LIN {X 0.066,Y -342.282,Z 1020.656,A 0.000,B 0.000,C 90.000,E1 118.103} C_DIS
LIN {X 0.176,Y -355.213,Z 1020.641,A 0.000,B 0.000,C 90.000,E1 115.335} C_DIS
LIN {X 0.119,Y -368.001,Z 1020.628,A 0.000,B 0.000,C 90.000,E1 112.950} C_DIS
LIN {X 0.098,Y -382.100,Z 1020.615,A 0.000,B 0.000,C 90.000,E1 110.610} C_DIS
LIN {X -0.206,Y -397.609,Z 1020.602,A 0.000,B 0.000,C 90.000,E1 108.362} C_DIS
LIN {X 0.126,Y -414.640,Z 1020.589,A 0.000,B 0.000,C 90.000,E1 106.079} C_DIS
LIN {X -0.157,Y -433.313,Z 1020.577,A 0.000,B 0.000,C 90.000,E1 103.939} C_DIS
LIN {X 0.189,Y -453.249,Z 1020.566,A 0.000,B 0.000,C 90.000,E1 101.827} C_DIS
LIN {X -0.120,Y -466.020,Z 1020.559,A 0.000,B 0.000,C 90.000,E1 100.658} C_DIS
LIN {X -0.093,Y -468.376,Z 1020.558,A 0.000,B 0.000,C 90.000,E1 100.423} C_DIS
LIN {X -0.148,Y -470.162,Z 1020.557,A 0.000,B 0.000,C 90.000,E1 100.197} C_DIS
LIN {X 0.167,Y -471.645,Z 1020.555,A 0.000,B 0.000,C 90.000,E1 99.905} C_DIS
LIN {X 0.018,Y -472.751,Z 1020.554,A 0.000,B 0.000,C 90.000,E1 99.670} C_DIS
LIN {X 0.125,Y -474.065,Z 1020.551,A 0.000,B 0.000,C 90.000,E1 99.151} C_DIS
LIN {X -0.156,Y -474.365,Z 1020.548,A 0.000,B 0.000,C 90.000,E1 98.681} C_DIS
LIN {X -0.034,Y -473.699,Z 1020.545,A 0.000,B 0.000,C 90.000,E1 98.163} C_DIS
LIN {X 0.093,Y -471.967,Z 1020.543,A 0.000,B 0.000,C 90.000,E1 97.644} C_DIS
LIN {X -0.049,Y -470.604,Z 1020.541,A 0.000,B 0.000,C 90.000,E1 97.409} C_DIS
LIN {X 0.009,Y -458.360,Z 1020.531,A 0.000,B 0.000,C 90.000,E1 95.625} C_DIS
LIN {X -0.178,Y -445.807,Z 1020.521,A 0.000,B 0.000,C 90.000,E1 93.841} C_DIS
LIN {X -0.035,Y -427.414,Z 1020.505,A 0.000,B 0.000,C 90.000,E1 90.917} C_DIS
LIN {X -0.048,Y -411.025,Z 1020.489,A 0.000,B 0.000,C 90.000,E1 87.936} C_DIS
LIN {X -0.010,Y -402.181,Z 1020.479,A 0.000,B 0.000,C 90.000,E1 86.274} C_DIS
LIN {X -0.112,Y -393.138,Z 1020.470,A 0.000,B 0.000,C 90.000,E1 84.609} C_DIS
LIN {X 0.091,Y -383.865,Z 1020.461,A 0.000,B 0.000,C 90.000,E1 82.875} C_DIS
LIN {X 0.119,Y -376.009,Z 1020.453,A 0.000,B 0.000,C 90.000,E1 81.432} C_DIS
LIN {X 0.047,Y -364.517,Z 1020.441,A 0.000,B 0.000,C 90.000,E1 79.398} C_DIS
LIN {X -0.187,Y -352.885,Z 1020.430,A 0.000,B 0.000,C 90.000,E1 77.353} C_DIS
LIN {X 0.067,Y -338.162,Z 1020.414,A 0.000,B 0.000,C 90.000,E1 74.574} C_DIS
LIN {X -0.175,Y -325.593,Z 1020.401,A 0.000,B 0.000,C 90.000,E1 72.127} C_DIS
LIN {X -0.035,Y -314.862,Z 1020.388,A 0.000,B 0.000,C 90.000,E1 69.880} C_DIS
LIN {X -0.110,Y -301.369,Z 1020.372,A 0.000,B 0.000,C 90.000,E1 66.975} C_DIS
LIN {X -0.154,Y -291.133,Z 1020.359,A 0.000,B 0.000,C 90.000,E1 64.665} C_DIS
LIN {X -0.052,Y -281.166,Z 1020.346,A 0.000,B 0.000,C 90.000,E1 62.281} C_DIS
LIN {X -0.099,Y -269.958,Z 1020.331,A 0.000,B 0.000,C 90.000,E1 59.537} C_DIS
LIN {X 0.078,Y -260.291,Z 1020.317,A 0.000,B 0.000,C 90.000,E1 57.041} C_DIS
LIN {X -0.018,Y -249.657,Z 1020.301,A 0.000,B 0.000,C 90.000,E1 54.196} C_DIS
LIN {X 0.045,Y -238.282,Z 1020.283,A 0.000,B 0.000,C 90.000,E1 50.884} C_DIS
LIN {X -0.116,Y -227.694,Z 1020.264,A 0.000,B 0.000,C 90.000,E1 47.553} C_DIS
LIN {X 0.123,Y -218.751,Z 1020.247,A 0.000,B 0.000,C 90.000,E1 44.433} C_DIS
LIN {X 0.004,Y -210.152,Z 1020.230,A 0.000,B 0.000,C 90.000,E1 41.353} C_DIS
LIN {X 0.040,Y -202.163,Z 1020.212,A 0.000,B 0.000,C 90.000,E1 38.177} C_DIS
LIN {X -0.039,Y -194.792,Z 1020.194,A 0.000,B 0.000,C 90.000,E1 34.978} C_DIS
LIN {X 0.070,Y -188.093,Z 1020.176,A 0.000,B 0.000,C 90.000,E1 31.671} C_DIS
LIN {X 0.036,Y -182.287,Z 1020.158,A 0.000,B 0.000,C 90.000,E1 28.359} C_DIS
LIN {X -0.071,Y -177.205,Z 1020.139,A 0.000,B 0.000,C 90.000,E1 25.027} C_DIS
LIN {X 0.031,Y -172.984,Z 1020.120,A 0.000,B 0.000,C 90.000,E1 21.589} C_DIS
LIN {X -0.060,Y -169.399,Z 1020.101,A 0.000,B 0.000,C 90.000,E1 18.181} C_DIS
LIN {X -0.011,Y -165.911,Z 1020.077,A 0.000,B 0.000,C 90.000,E1 13.828} C_DIS
LIN {X 0.025,Y -163.211,Z 1020.048,A 0.000,B 0.000,C 90.000,E1 8.568} C_DIS
LIN {X 0.015,Y -164.093,Z 1019.953,A 0.000,B 0.000,C 90.000,E1 351.602} C_DIS
LIN {X 0.009,Y -167.296,Z 1019.924,A 0.000,B 0.000,C 90.000,E1 346.353} C_DIS
LIN {X 0.037,Y -171.068,Z 1019.900,A 0.000,B 0.000,C 90.000,E1 342.000} C_DIS
LIN {X -0.079,Y -174.981,Z 1019.881,A 0.000,B 0.000,C 90.000,E1 338.592} C_DIS
LIN {X -0.001,Y -179.715,Z 1019.862,A 0.000,B 0.000,C 90.000,E1 335.153} C_DIS
LIN {X 0.024,Y -185.257,Z 1019.843,A 0.000,B 0.000,C 90.000,E1 331.769} C_DIS
LIN {X -0.041,Y -191.575,Z 1019.825,A 0.000,B 0.000,C 90.000,E1 328.456} C_DIS
LIN {X -0.078,Y -198.576,Z 1019.806,A 0.000,B 0.000,C 90.000,E1 325.182} C_DIS
LIN {X -0.040,Y -207.196,Z 1019.786,A 0.000,B 0.000,C 90.000,E1 321.537} C_DIS
LIN {X 0.037,Y -216.493,Z 1019.766,A 0.000,B 0.000,C 90.000,E1 317.957} C_DIS
LIN {X 0.107,Y -225.454,Z 1019.749,A 0.000,B 0.000,C 90.000,E1 314.838} C_DIS
LIN {X -0.021,Y -234.071,Z 1019.734,A 0.000,B 0.000,C 90.000,E1 312.204} C_DIS
LIN {X 0.094,Y -242.569,Z 1019.722,A 0.000,B 0.000,C 90.000,E1 309.930} C_DIS
LIN {X 0.056,Y -248.911,Z 1019.714,A 0.000,B 0.000,C 90.000,E1 308.463} C_DIS
LIN {X -0.034,Y -257.706,Z 1019.704,A 0.000,B 0.000,C 90.000,E1 306.664} C_DIS
LIN {X -0.168,Y -271.393,Z 1019.690,A 0.000,B 0.000,C 90.000,E1 304.199} C_DIS
LIN {X 0.040,Y -288.410,Z 1019.674,A 0.000,B 0.000,C 90.000,E1 301.386} C_DIS
LIN {X 0.130,Y -309.092,Z 1019.658,A 0.000,B 0.000,C 90.000,E1 298.359} C_DIS
LIN {X 0.007,Y -324.070,Z 1019.647,A 0.000,B 0.000,C 90.000,E1 296.437} C_DIS
LIN {X -0.043,Y -337.092,Z 1019.639,A 0.000,B 0.000,C 90.000,E1 294.951} C_DIS
LIN {X -0.147,Y -364.351,Z 1019.623,A 0.000,B 0.000,C 90.000,E1 292.206} C_DIS
LIN {X -0.138,Y -383.717,Z 1019.613,A 0.000,B 0.000,C 90.000,E1 290.429} C_DIS
LIN {X 0.093,Y -402.310,Z 1019.604,A 0.000,B 0.000,C 90.000,E1 288.725} C_DIS
LIN {X 0.012,Y -412.772,Z 1019.599,A 0.000,B 0.000,C 90.000,E1 287.764} C_DIS
LIN {X -0.146,Y -420.410,Z 1019.595,A 0.000,B 0.000,C 90.000,E1 287.040} C_DIS
LIN {X -0.161,Y -427.896,Z 1019.590,A 0.000,B 0.000,C 90.000,E1 286.260} C_DIS
LIN {X -0.164,Y -437.601,Z 1019.584,A 0.000,B 0.000,C 90.000,E1 285.190} C_DIS
LIN {X -0.089,Y -446.673,Z 1019.578,A 0.000,B 0.000,C 90.000,E1 284.120} C_DIS
LIN {X -0.014,Y -455.104,Z 1019.573,A 0.000,B 0.000,C 90.000,E1 283.063} C_DIS
LIN {X -0.114,Y -460.826,Z 1019.568,A 0.000,B 0.000,C 90.000,E1 282.299} C_DIS
LIN {X -0.161,Y -466.044,Z 1019.564,A 0.000,B 0.000,C 90.000,E1 281.535} C_DIS
LIN {X -0.261,Y -470.809,Z 1019.560,A 0.000,B 0.000,C 90.000,E1 280.782} C_DIS
LIN {X 0.241,Y -474.949,Z 1019.555,A 0.000,B 0.000,C 90.000,E1 279.962} C_DIS
LIN {X 0.228,Y -478.512,Z 1019.551,A 0.000,B 0.000,C 90.000,E1 279.208} C_DIS
LIN {X -0.101,Y -480.580,Z 1019.549,A 0.000,B 0.000,C 90.000,E1 278.746} C_DIS
LIN {X 0.128,Y -482.342,Z 1019.546,A 0.000,B 0.000,C 90.000,E1 278.219} C_DIS
LIN {X -0.010,Y -485.160,Z 1019.540,A 0.000,B 0.000,C 90.000,E1 277.239} C_DIS
LIN {X 0.176,Y -486.261,Z 1019.537,A 0.000,B 0.000,C 90.000,E1 276.720} C_DIS
LIN {X -0.113,Y -487.145,Z 1019.535,A 0.000,B 0.000,C 90.000,E1 276.258} C_DIS
LIN {X 0.088,Y -487.739,Z 1019.532,A 0.000,B 0.000,C 90.000,E1 275.739} C_DIS
LIN {X -0.193,Y -487.996,Z 1019.529,A 0.000,B 0.000,C 90.000,E1 275.277} C_DIS
LIN {X 0.015,Y -487.823,Z 1019.526,A 0.000,B 0.000,C 90.000,E1 274.759} C_DIS
LIN {X 0.184,Y -487.214,Z 1019.524,A 0.000,B 0.000,C 90.000,E1 274.245} C_DIS
LIN {X -0.096,Y -486.033,Z 1019.521,A 0.000,B 0.000,C 90.000,E1 273.784} C_DIS
LIN {X 0.075,Y -484.262,Z 1019.518,A 0.000,B 0.000,C 90.000,E1 273.269} C_DIS
LIN {X -0.216,Y -481.851,Z 1019.515,A 0.000,B 0.000,C 90.000,E1 272.808} C_DIS
LIN {X -0.066,Y -478.743,Z 1019.513,A 0.000,B 0.000,C 90.000,E1 272.293} C_DIS
LIN {X 0.085,Y -474.804,Z 1019.510,A 0.000,B 0.000,C 90.000,E1 271.776} C_DIS
LIN {X 0.197,Y -469.936,Z 1019.507,A 0.000,B 0.000,C 90.000,E1 271.260} C_DIS
LIN {X 0.068,Y -467.256,Z 1019.506,A 0.000,B 0.000,C 90.000,E1 271.031} C_DIS
LIN {X 0.036,Y -461.351,Z 1019.503,A 0.000,B 0.000,C 90.000,E1 270.573} C_DIS
LIN {X -0.003,Y -455.012,Z 1019.501,A 0.000,B 0.000,C 90.000,E1 270.172} C_DIS
LIN {X -0.134,Y -451.585,Z 1019.500,A 0.000,B 0.000,C 90.000,E1 270.000} C_DIS
LIN {X 0.031,Y -444.187,Z 1019.498,A 0.000,B 0.000,C 90.000,E1 269.656} C_DIS
LIN {X -0.142,Y -436.615,Z 1019.497,A 0.000,B 0.000,C 90.000,E1 269.427} C_DIS
LIN {X 0.122,Y -428.268,Z 1019.496,A 0.000,B 0.000,C 90.000,E1 269.198} C_DIS
LIN {X -0.012,Y -419.507,Z 1019.495,A 0.000,B 0.000,C 90.000,E1 269.083} C_DIS
LIN {X 0.127,Y -409.897,Z 1019.494,A 0.000,B 0.000,C 90.000,E1 268.969} C_DIS
LIN {X 0.140,Y -400.201,Z 1019.494,A 0.000,B 0.000,C 90.000,E1 268.912} C_DIS
LIN {X 0.034,Y -181.301,Z 1019.494,A 0.000,B 0.000,C 90.000,E1 268.912} C_DIS
LIN {X -0.096,Y -180.897,Z 1019.473,A 0.000,B 0.000,C 90.000,E1 265.241} C_DIS
LIN {X -0.073,Y -179.844,Z 1019.459,A 0.000,B 0.000,C 90.000,E1 262.704} C_DIS
LIN {X -0.016,Y -179.028,Z 1019.445,A 0.000,B 0.000,C 90.000,E1 260.151} C_DIS
LIN {X 0.046,Y -178.676,Z 1019.441,A 0.000,B 0.000,C 90.000,E1 259.285} C_DIS
LIN {X -0.018,Y -175.725,Z 1019.412,A 0.000,B 0.000,C 90.000,E1 254.212} C_DIS
LIN {X -0.002,Y -172.442,Z 1019.388,A 0.000,B 0.000,C 90.000,E1 249.934} C_DIS
LIN {X -0.046,Y -171.274,Z 1019.379,A 0.000,B 0.000,C 90.000,E1 248.230} C_DIS
LIN {X 0.000,Y -167.543,Z 1019.355,A 0.000,B 0.000,C 90.000,E1 243.896} C_DIS
LIN {X 0.014,Y -166.160,Z 1019.345,A 0.000,B 0.000,C 90.000,E1 242.153} C_DIS
LIN {X 0.004,Y -162.935,Z 1019.326,A 0.000,B 0.000,C 90.000,E1 238.663} C_DIS
LIN {X -0.019,Y -161.606,Z 1019.316,A 0.000,B 0.000,C 90.000,E1 236.914} C_DIS
LIN {X -0.043,Y -159.132,Z 1019.301,A 0.000,B 0.000,C 90.000,E1 234.276} C_DIS
LIN {X -0.032,Y -155.653,Z 1019.277,A 0.000,B 0.000,C 90.000,E1 229.828} C_DIS
LIN {X 0.020,Y -151.924,Z 1019.252,A 0.000,B 0.000,C 90.000,E1 225.324} C_DIS
LIN {X 0.036,Y -150.160,Z 1019.237,A 0.000,B 0.000,C 90.000,E1 222.609} C_DIS
LIN {X -0.044,Y -146.939,Z 1019.212,A 0.000,B 0.000,C 90.000,E1 218.096} C_DIS
LIN {X 0.062,Y -145.527,Z 1019.196,A 0.000,B 0.000,C 90.000,E1 215.311} C_DIS
LIN {X -0.017,Y -142.926,Z 1019.171,A 0.000,B 0.000,C 90.000,E1 210.747} C_DIS
LIN {X -0.018,Y -141.549,Z 1019.150,A 0.000,B 0.000,C 90.000,E1 207.052} C_DIS
LIN {X -0.028,Y -139.405,Z 1019.114,A 0.000,B 0.000,C 90.000,E1 200.556} C_DIS
LIN {X 0.026,Y -139.123,Z 1019.104,A 0.000,B 0.000,C 90.000,E1 198.671} C_DIS
LIN {X 0.057,Y -138.352,Z 1019.057,A 0.000,B 0.000,C 90.000,E1 190.254} C_DIS
LIN {X 0.047,Y -139.502,Z 1019.005,A 0.000,B 0.000,C 90.000,E1 180.917} C_DIS
LIN {X -0.012,Y -141.130,Z 1018.974,A 0.000,B 0.000,C 90.000,E1 175.355} C_DIS
LIN {X -0.058,Y -142.510,Z 1018.959,A 0.000,B 0.000,C 90.000,E1 172.591} C_DIS
LIN {X 0.029,Y -144.770,Z 1018.933,A 0.000,B 0.000,C 90.000,E1 167.937} C_DIS
LIN {X -0.021,Y -147.382,Z 1018.913,A 0.000,B 0.000,C 90.000,E1 164.283} C_DIS
LIN {X 0.041,Y -150.712,Z 1018.887,A 0.000,B 0.000,C 90.000,E1 159.699} C_DIS
LIN {X -0.019,Y -154.192,Z 1018.867,A 0.000,B 0.000,C 90.000,E1 156.102} C_DIS
LIN {X 0.050,Y -157.631,Z 1018.847,A 0.000,B 0.000,C 90.000,E1 152.487} C_DIS
LIN {X -0.002,Y -161.888,Z 1018.828,A 0.000,B 0.000,C 90.000,E1 148.948} C_DIS
LIN {X -0.029,Y -166.078,Z 1018.808,A 0.000,B 0.000,C 90.000,E1 145.435} C_DIS
LIN {X -0.029,Y -171.085,Z 1018.789,A 0.000,B 0.000,C 90.000,E1 141.949} C_DIS
LIN {X 0.026,Y -175.959,Z 1018.769,A 0.000,B 0.000,C 90.000,E1 138.485} C_DIS
LIN {X -0.114,Y -180.202,Z 1018.755,A 0.000,B 0.000,C 90.000,E1 135.972} C_DIS
LIN {X 0.116,Y -185.618,Z 1018.736,A 0.000,B 0.000,C 90.000,E1 132.528} C_DIS
LIN {X -0.099,Y -190.213,Z 1018.723,A 0.000,B 0.000,C 90.000,E1 130.092} C_DIS
LIN {X 0.100,Y -196.811,Z 1018.702,A 0.000,B 0.000,C 90.000,E1 126.297} C_DIS
LIN {X 0.094,Y -302.042,Z 1018.702,A 0.000,B 0.000,C 90.000,E1 126.297} C_DIS
LIN {X -0.088,Y -303.802,Z 1018.702,A 0.000,B 0.000,C 90.000,E1 126.297} C_DIS
LIN {X 0.096,Y -309.635,Z 1018.700,A 0.000,B 0.000,C 90.000,E1 125.931} C_DIS
LIN {X 0.013,Y -312.804,Z 1018.698,A 0.000,B 0.000,C 90.000,E1 125.598} C_DIS
LIN {X -0.073,Y -314.784,Z 1018.696,A 0.000,B 0.000,C 90.000,E1 125.311} C_DIS
LIN {X -0.160,Y -316.338,Z 1018.694,A 0.000,B 0.000,C 90.000,E1 125.025} C_DIS
LIN {X -0.099,Y -317.652,Z 1018.693,A 0.000,B 0.000,C 90.000,E1 124.692} C_DIS
LIN {X 0.112,Y -328.633,Z 1018.675,A 0.000,B 0.000,C 90.000,E1 121.465} C_DIS
LIN {X -0.151,Y -339.864,Z 1018.659,A 0.000,B 0.000,C 90.000,E1 118.693} C_DIS
LIN {X 0.041,Y -352.501,Z 1018.644,A 0.000,B 0.000,C 90.000,E1 115.899} C_DIS
LIN {X -0.024,Y -366.663,Z 1018.629,A 0.000,B 0.000,C 90.000,E1 113.206} C_DIS
LIN {X -0.081,Y -380.628,Z 1018.616,A 0.000,B 0.000,C 90.000,E1 110.865} C_DIS
LIN {X 0.082,Y -395.995,Z 1018.603,A 0.000,B 0.000,C 90.000,E1 108.544} C_DIS
LIN {X -0.011,Y -412.870,Z 1018.591,A 0.000,B 0.000,C 90.000,E1 106.315} C_DIS
LIN {X 0.075,Y -431.376,Z 1018.578,A 0.000,B 0.000,C 90.000,E1 104.120} C_DIS
LIN {X -0.142,Y -451.247,Z 1018.567,A 0.000,B 0.000,C 90.000,E1 102.063} C_DIS
LIN {X -0.071,Y -466.541,Z 1018.559,A 0.000,B 0.000,C 90.000,E1 100.602} C_DIS
LIN {X -0.038,Y -468.778,Z 1018.558,A 0.000,B 0.000,C 90.000,E1 100.366} C_DIS
LIN {X -0.089,Y -470.466,Z 1018.556,A 0.000,B 0.000,C 90.000,E1 100.141} C_DIS
LIN {X -0.237,Y -471.872,Z 1018.555,A 0.000,B 0.000,C 90.000,E1 99.905} C_DIS
LIN {X 0.079,Y -472.917,Z 1018.553,A 0.000,B 0.000,C 90.000,E1 99.613} C_DIS
LIN {X 0.189,Y -474.131,Z 1018.551,A 0.000,B 0.000,C 90.000,E1 99.095} C_DIS
LIN {X -0.090,Y -474.342,Z 1018.548,A 0.000,B 0.000,C 90.000,E1 98.624} C_DIS
LIN {X 0.034,Y -473.586,Z 1018.545,A 0.000,B 0.000,C 90.000,E1 98.106} C_DIS
LIN {X 0.160,Y -471.744,Z 1018.542,A 0.000,B 0.000,C 90.000,E1 97.587} C_DIS
LIN {X 0.018,Y -470.307,Z 1018.541,A 0.000,B 0.000,C 90.000,E1 97.352} C_DIS
LIN {X 0.071,Y -458.038,Z 1018.531,A 0.000,B 0.000,C 90.000,E1 95.568} C_DIS
LIN {X -0.124,Y -445.510,Z 1018.521,A 0.000,B 0.000,C 90.000,E1 93.784} C_DIS
LIN {X 0.009,Y -427.148,Z 1018.505,A 0.000,B 0.000,C 90.000,E1 90.859} C_DIS
LIN {X -0.100,Y -412.218,Z 1018.490,A 0.000,B 0.000,C 90.000,E1 88.165} C_DIS
LIN {X -0.036,Y -403.421,Z 1018.481,A 0.000,B 0.000,C 90.000,E1 86.502} C_DIS
LIN {X -0.112,Y -394.391,Z 1018.471,A 0.000,B 0.000,C 90.000,E1 84.837} C_DIS
LIN {X 0.072,Y -385.151,Z 1018.462,A 0.000,B 0.000,C 90.000,E1 83.109} C_DIS
LIN {X 0.165,Y -377.327,Z 1018.454,A 0.000,B 0.000,C 90.000,E1 81.659} C_DIS
LIN {X 0.067,Y -365.865,Z 1018.442,A 0.000,B 0.000,C 90.000,E1 79.634} C_DIS
LIN {X -0.147,Y -354.256,Z 1018.431,A 0.000,B 0.000,C 90.000,E1 77.589} C_DIS
LIN {X 0.147,Y -339.465,Z 1018.416,A 0.000,B 0.000,C 90.000,E1 74.810} C_DIS
LIN {X -0.066,Y -326.902,Z 1018.402,A 0.000,B 0.000,C 90.000,E1 72.362} C_DIS
LIN {X 0.098,Y -316.133,Z 1018.390,A 0.000,B 0.000,C 90.000,E1 70.115} C_DIS
LIN {X 0.042,Y -304.041,Z 1018.375,A 0.000,B 0.000,C 90.000,E1 67.539} C_DIS
LIN {X 0.051,Y -293.785,Z 1018.362,A 0.000,B 0.000,C 90.000,E1 65.229} C_DIS
LIN {X 0.049,Y -282.339,Z 1018.347,A 0.000,B 0.000,C 90.000,E1 62.538} C_DIS
LIN {X 0.086,Y -272.484,Z 1018.334,A 0.000,B 0.000,C 90.000,E1 60.127} C_DIS
LIN {X -0.046,Y -262.771,Z 1018.321,A 0.000,B 0.000,C 90.000,E1 57.709} C_DIS
LIN {X 0.012,Y -250.699,Z 1018.303,A 0.000,B 0.000,C 90.000,E1 54.482} C_DIS
LIN {X 0.107,Y -239.244,Z 1018.284,A 0.000,B 0.000,C 90.000,E1 51.170} C_DIS
LIN {X -0.032,Y -228.592,Z 1018.266,A 0.000,B 0.000,C 90.000,E1 47.838} C_DIS
LIN {X -0.003,Y -218.486,Z 1018.247,A 0.000,B 0.000,C 90.000,E1 44.393} C_DIS
LIN {X 0.026,Y -209.894,Z 1018.229,A 0.000,B 0.000,C 90.000,E1 41.272} C_DIS
LIN {X 0.054,Y -201.898,Z 1018.212,A 0.000,B 0.000,C 90.000,E1 38.096} C_DIS
LIN {X -0.034,Y -194.521,Z 1018.194,A 0.000,B 0.000,C 90.000,E1 34.898} C_DIS
LIN {X 0.066,Y -187.851,Z 1018.176,A 0.000,B 0.000,C 90.000,E1 31.592} C_DIS
LIN {X 0.022,Y -182.087,Z 1018.157,A 0.000,B 0.000,C 90.000,E1 28.281} C_DIS
LIN {X 0.065,Y -177.024,Z 1018.138,A 0.000,B 0.000,C 90.000,E1 24.899} C_DIS
LIN {X -0.065,Y -172.823,Z 1018.120,A 0.000,B 0.000,C 90.000,E1 21.535} C_DIS
LIN {X 0.059,Y -169.266,Z 1018.100,A 0.000,B 0.000,C 90.000,E1 18.055} C_DIS
LIN {X 0.057,Y -165.790,Z 1018.076,A 0.000,B 0.000,C 90.000,E1 13.716} C_DIS
LIN {X -0.068,Y -163.126,Z 1018.047,A 0.000,B 0.000,C 90.000,E1 8.511} C_DIS
LIN {X 0.045,Y -163.647,Z 1017.958,A 0.000,B 0.000,C 90.000,E1 352.470} C_DIS
LIN {X -0.004,Y -166.615,Z 1017.929,A 0.000,B 0.000,C 90.000,E1 347.229} C_DIS
LIN {X -0.088,Y -170.202,Z 1017.905,A 0.000,B 0.000,C 90.000,E1 342.906} C_DIS
LIN {X -0.064,Y -173.890,Z 1017.886,A 0.000,B 0.000,C 90.000,E1 339.444} C_DIS
LIN {X 0.010,Y -178.448,Z 1017.867,A 0.000,B 0.000,C 90.000,E1 335.997} C_DIS
LIN {X -0.002,Y -183.796,Z 1017.848,A 0.000,B 0.000,C 90.000,E1 332.615} C_DIS
LIN {X -0.038,Y -189.938,Z 1017.829,A 0.000,B 0.000,C 90.000,E1 329.282} C_DIS
LIN {X 0.045,Y -196.801,Z 1017.811,A 0.000,B 0.000,C 90.000,E1 325.960} C_DIS
LIN {X 0.033,Y -204.261,Z 1017.793,A 0.000,B 0.000,C 90.000,E1 322.718} C_DIS
LIN {X 0.022,Y -213.342,Z 1017.773,A 0.000,B 0.000,C 90.000,E1 319.138} C_DIS
LIN {X -0.129,Y -221.985,Z 1017.756,A 0.000,B 0.000,C 90.000,E1 316.053} C_DIS
LIN {X 0.086,Y -231.473,Z 1017.739,A 0.000,B 0.000,C 90.000,E1 312.933} C_DIS
LIN {X 0.005,Y -238.160,Z 1017.728,A 0.000,B 0.000,C 90.000,E1 311.067} C_DIS
LIN {X 0.055,Y -245.632,Z 1017.718,A 0.000,B 0.000,C 90.000,E1 309.197} C_DIS
LIN {X -0.065,Y -255.876,Z 1017.706,A 0.000,B 0.000,C 90.000,E1 307.030} C_DIS
LIN {X -0.147,Y -267.382,Z 1017.694,A 0.000,B 0.000,C 90.000,E1 304.898} C_DIS
LIN {X -0.042,Y -284.125,Z 1017.678,A 0.000,B 0.000,C 90.000,E1 302.084} C_DIS
LIN {X 0.072,Y -304.377,Z 1017.661,A 0.000,B 0.000,C 90.000,E1 299.027} C_DIS
LIN {X 0.075,Y -321.573,Z 1017.649,A 0.000,B 0.000,C 90.000,E1 296.744} C_DIS
LIN {X 0.177,Y -334.532,Z 1017.640,A 0.000,B 0.000,C 90.000,E1 295.207} C_DIS
LIN {X -0.085,Y -353.579,Z 1017.629,A 0.000,B 0.000,C 90.000,E1 293.259} C_DIS
LIN {X -0.079,Y -381.144,Z 1017.615,A 0.000,B 0.000,C 90.000,E1 290.663} C_DIS
LIN {X 0.244,Y -397.458,Z 1017.607,A 0.000,B 0.000,C 90.000,E1 289.141} C_DIS
LIN {X 0.186,Y -408.135,Z 1017.601,A 0.000,B 0.000,C 90.000,E1 288.181} C_DIS
LIN {X -0.013,Y -418.408,Z 1017.596,A 0.000,B 0.000,C 90.000,E1 287.221} C_DIS
LIN {X 0.043,Y -425.893,Z 1017.591,A 0.000,B 0.000,C 90.000,E1 286.441} C_DIS
LIN {X 0.058,Y -435.650,Z 1017.585,A 0.000,B 0.000,C 90.000,E1 285.371} C_DIS
LIN {X 0.116,Y -444.869,Z 1017.580,A 0.000,B 0.000,C 90.000,E1 284.300} C_DIS
LIN {X 0.176,Y -453.397,Z 1017.574,A 0.000,B 0.000,C 90.000,E1 283.244} C_DIS
LIN {X 0.071,Y -459.302,Z 1017.569,A 0.000,B 0.000,C 90.000,E1 282.479} C_DIS
LIN {X -0.151,Y -466.373,Z 1017.564,A 0.000,B 0.000,C 90.000,E1 281.478} C_DIS
LIN {X -0.158,Y -471.093,Z 1017.559,A 0.000,B 0.000,C 90.000,E1 280.715} C_DIS
LIN {X -0.208,Y -475.240,Z 1017.555,A 0.000,B 0.000,C 90.000,E1 279.962} C_DIS
LIN {X -0.222,Y -478.787,Z 1017.551,A 0.000,B 0.000,C 90.000,E1 279.208} C_DIS
LIN {X -0.003,Y -480.860,Z 1017.548,A 0.000,B 0.000,C 90.000,E1 278.681} C_DIS
LIN {X 0.155,Y -482.595,Z 1017.545,A 0.000,B 0.000,C 90.000,E1 278.163} C_DIS
LIN {X -0.157,Y -484.088,Z 1017.543,A 0.000,B 0.000,C 90.000,E1 277.701} C_DIS
LIN {X 0.022,Y -485.362,Z 1017.540,A 0.000,B 0.000,C 90.000,E1 277.182} C_DIS
LIN {X 0.210,Y -486.445,Z 1017.537,A 0.000,B 0.000,C 90.000,E1 276.663} C_DIS
LIN {X -0.078,Y -487.302,Z 1017.534,A 0.000,B 0.000,C 90.000,E1 276.201} C_DIS
LIN {X 0.125,Y -487.917,Z 1017.532,A 0.000,B 0.000,C 90.000,E1 275.682} C_DIS
LIN {X -0.155,Y -488.131,Z 1017.529,A 0.000,B 0.000,C 90.000,E1 275.220} C_DIS
LIN {X 0.053,Y -487.921,Z 1017.526,A 0.000,B 0.000,C 90.000,E1 274.702} C_DIS
LIN {X 0.225,Y -487.271,Z 1017.523,A 0.000,B 0.000,C 90.000,E1 274.188} C_DIS
LIN {X -0.055,Y -486.048,Z 1017.521,A 0.000,B 0.000,C 90.000,E1 273.726} C_DIS
LIN {X 0.117,Y -484.256,Z 1017.518,A 0.000,B 0.000,C 90.000,E1 273.212} C_DIS
LIN {X -0.175,Y -481.819,Z 1017.515,A 0.000,B 0.000,C 90.000,E1 272.751} C_DIS
LIN {X -0.024,Y -478.629,Z 1017.512,A 0.000,B 0.000,C 90.000,E1 272.236} C_DIS
LIN {X 0.125,Y -474.612,Z 1017.510,A 0.000,B 0.000,C 90.000,E1 271.718} C_DIS
LIN {X 0.236,Y -469.684,Z 1017.507,A 0.000,B 0.000,C 90.000,E1 271.203} C_DIS
LIN {X -0.005,Y -463.904,Z 1017.504,A 0.000,B 0.000,C 90.000,E1 270.745} C_DIS
LIN {X 0.213,Y -457.674,Z 1017.502,A 0.000,B 0.000,C 90.000,E1 270.286} C_DIS
LIN {X -0.012,Y -451.050,Z 1017.500,A 0.000,B 0.000,C 90.000,E1 269.943} C_DIS
LIN {X -0.212,Y -443.741,Z 1017.498,A 0.000,B 0.000,C 90.000,E1 269.656} C_DIS
LIN {X 0.132,Y -436.315,Z 1017.497,A 0.000,B 0.000,C 90.000,E1 269.370} C_DIS
LIN {X 0.010,Y -428.264,Z 1017.496,A 0.000,B 0.000,C 90.000,E1 269.198} C_DIS
LIN {X -0.135,Y -419.304,Z 1017.495,A 0.000,B 0.000,C 90.000,E1 269.083} C_DIS
LIN {X 0.009,Y -409.433,Z 1017.494,A 0.000,B 0.000,C 90.000,E1 268.969} C_DIS
LIN {X 0.031,Y -399.434,Z 1017.494,A 0.000,B 0.000,C 90.000,E1 268.912} C_DIS
LIN {X -0.014,Y -181.298,Z 1017.494,A 0.000,B 0.000,C 90.000,E1 268.912} C_DIS
LIN {X 0.050,Y -180.895,Z 1017.473,A 0.000,B 0.000,C 90.000,E1 265.179} C_DIS
LIN {X 0.057,Y -179.837,Z 1017.459,A 0.000,B 0.000,C 90.000,E1 262.648} C_DIS
LIN {X -0.064,Y -179.024,Z 1017.445,A 0.000,B 0.000,C 90.000,E1 260.151} C_DIS
LIN {X -0.002,Y -178.665,Z 1017.440,A 0.000,B 0.000,C 90.000,E1 259.285} C_DIS
LIN {X -0.065,Y -175.716,Z 1017.412,A 0.000,B 0.000,C 90.000,E1 254.212} C_DIS
LIN {X -0.049,Y -172.431,Z 1017.388,A 0.000,B 0.000,C 90.000,E1 249.934} C_DIS
LIN {X -0.030,Y -171.258,Z 1017.379,A 0.000,B 0.000,C 90.000,E1 248.209} C_DIS
LIN {X -0.046,Y -167.531,Z 1017.355,A 0.000,B 0.000,C 90.000,E1 243.896} C_DIS
LIN {X 0.036,Y -166.925,Z 1017.350,A 0.000,B 0.000,C 90.000,E1 242.999} C_DIS
LIN {X -0.042,Y -162.922,Z 1017.326,A 0.000,B 0.000,C 90.000,E1 238.663} C_DIS
LIN {X -0.064,Y -161.595,Z 1017.316,A 0.000,B 0.000,C 90.000,E1 236.914} C_DIS
LIN {X 0.062,Y -158.337,Z 1017.296,A 0.000,B 0.000,C 90.000,E1 233.336} C_DIS
LIN {X -0.076,Y -155.640,Z 1017.277,A 0.000,B 0.000,C 90.000,E1 229.828} C_DIS
LIN {X -0.024,Y -151.913,Z 1017.252,A 0.000,B 0.000,C 90.000,E1 225.324} C_DIS
LIN {X -0.008,Y -150.145,Z 1017.237,A 0.000,B 0.000,C 90.000,E1 222.609} C_DIS
LIN {X -0.087,Y -146.930,Z 1017.211,A 0.000,B 0.000,C 90.000,E1 218.096} C_DIS
LIN {X 0.020,Y -145.517,Z 1017.196,A 0.000,B 0.000,C 90.000,E1 215.311} C_DIS
LIN {X 0.014,Y -142.918,Z 1017.171,A 0.000,B 0.000,C 90.000,E1 210.718} C_DIS
LIN {X 0.067,Y -141.540,Z 1017.150,A 0.000,B 0.000,C 90.000,E1 207.001} C_DIS
LIN {X -0.021,Y -139.402,Z 1017.114,A 0.000,B 0.000,C 90.000,E1 200.536} C_DIS
LIN {X -0.016,Y -139.118,Z 1017.104,A 0.000,B 0.000,C 90.000,E1 198.671} C_DIS
LIN {X 0.016,Y -138.352,Z 1017.057,A 0.000,B 0.000,C 90.000,E1 190.254} C_DIS
LIN {X 0.006,Y -139.504,Z 1017.005,A 0.000,B 0.000,C 90.000,E1 180.917} C_DIS
LIN {X -0.053,Y -141.138,Z 1016.974,A 0.000,B 0.000,C 90.000,E1 175.355} C_DIS
LIN {X 0.041,Y -142.518,Z 1016.959,A 0.000,B 0.000,C 90.000,E1 172.534} C_DIS
LIN {X -0.014,Y -144.780,Z 1016.933,A 0.000,B 0.000,C 90.000,E1 167.937} C_DIS
LIN {X -0.025,Y -147.395,Z 1016.913,A 0.000,B 0.000,C 90.000,E1 164.267} C_DIS
LIN {X -0.003,Y -150.726,Z 1016.887,A 0.000,B 0.000,C 90.000,E1 159.699} C_DIS
LIN {X -0.063,Y -154.208,Z 1016.867,A 0.000,B 0.000,C 90.000,E1 156.102} C_DIS
LIN {X 0.005,Y -157.648,Z 1016.847,A 0.000,B 0.000,C 90.000,E1 152.487} C_DIS
LIN {X -0.048,Y -161.908,Z 1016.827,A 0.000,B 0.000,C 90.000,E1 148.948} C_DIS
LIN {X 0.061,Y -166.099,Z 1016.808,A 0.000,B 0.000,C 90.000,E1 145.388} C_DIS
LIN {X 0.059,Y -171.108,Z 1016.788,A 0.000,B 0.000,C 90.000,E1 141.904} C_DIS
LIN {X -0.022,Y -175.983,Z 1016.769,A 0.000,B 0.000,C 90.000,E1 138.485} C_DIS
LIN {X 0.093,Y -180.229,Z 1016.755,A 0.000,B 0.000,C 90.000,E1 135.891} C_DIS
LIN {X 0.066,Y -185.644,Z 1016.736,A 0.000,B 0.000,C 90.000,E1 132.528} C_DIS
LIN {X 0.120,Y -190.243,Z 1016.722,A 0.000,B 0.000,C 90.000,E1 130.011} C_DIS
LIN {X -0.044,Y -196.738,Z 1016.702,A 0.000,B 0.000,C 90.000,E1 126.377} C_DIS
LIN {X -0.102,Y -301.851,Z 1016.702,A 0.000,B 0.000,C 90.000,E1 126.377} C_DIS
LIN {X 0.082,Y -304.015,Z 1016.702,A 0.000,B 0.000,C 90.000,E1 126.297} C_DIS
LIN {X -0.075,Y -307.808,Z 1016.701,A 0.000,B 0.000,C 90.000,E1 126.137} C_DIS
LIN {X 0.016,Y -310.102,Z 1016.700,A 0.000,B 0.000,C 90.000,E1 125.931} C_DIS
LIN {X 0.071,Y -313.964,Z 1016.697,A 0.000,B 0.000,C 90.000,E1 125.438} C_DIS
LIN {X 0.115,Y -315.769,Z 1016.695,A 0.000,B 0.000,C 90.000,E1 125.105} C_DIS
LIN {X -0.097,Y -317.181,Z 1016.693,A 0.000,B 0.000,C 90.000,E1 124.818} C_DIS
LIN {X 0.203,Y -329.323,Z 1016.674,A 0.000,B 0.000,C 90.000,E1 121.258} C_DIS
LIN {X -0.041,Y -340.646,Z 1016.658,A 0.000,B 0.000,C 90.000,E1 118.487} C_DIS
LIN {X 0.016,Y -353.382,Z 1016.643,A 0.000,B 0.000,C 90.000,E1 115.720} C_DIS
LIN {X -0.018,Y -367.649,Z 1016.628,A 0.000,B 0.000,C 90.000,E1 113.025} C_DIS
LIN {X 0.090,Y -381.718,Z 1016.615,A 0.000,B 0.000,C 90.000,E1 110.663} C_DIS
LIN {X 0.147,Y -397.193,Z 1016.602,A 0.000,B 0.000,C 90.000,E1 108.362} C_DIS
LIN {X 0.086,Y -414.187,Z 1016.590,A 0.000,B 0.000,C 90.000,E1 106.134} C_DIS
LIN {X 0.102,Y -432.822,Z 1016.578,A 0.000,B 0.000,C 90.000,E1 103.953} C_DIS
LIN {X 0.082,Y -452.757,Z 1016.566,A 0.000,B 0.000,C 90.000,E1 101.883} C_DIS
LIN {X 0.148,Y -467.967,Z 1016.558,A 0.000,B 0.000,C 90.000,E1 100.433} C_DIS
LIN {X 0.111,Y -469.908,Z 1016.557,A 0.000,B 0.000,C 90.000,E1 100.197} C_DIS
LIN {X 0.071,Y -471.382,Z 1016.555,A 0.000,B 0.000,C 90.000,E1 99.962} C_DIS
LIN {X 0.168,Y -473.407,Z 1016.553,A 0.000,B 0.000,C 90.000,E1 99.443} C_DIS
LIN {X -0.118,Y -474.298,Z 1016.550,A 0.000,B 0.000,C 90.000,E1 98.973} C_DIS
LIN {X 0.001,Y -474.212,Z 1016.547,A 0.000,B 0.000,C 90.000,E1 98.454} C_DIS
LIN {X 0.128,Y -473.140,Z 1016.544,A 0.000,B 0.000,C 90.000,E1 97.936} C_DIS
LIN {X -0.011,Y -472.189,Z 1016.543,A 0.000,B 0.000,C 90.000,E1 97.701} C_DIS
LIN {X -0.151,Y -470.900,Z 1016.541,A 0.000,B 0.000,C 90.000,E1 97.466} C_DIS
LIN {X 0.133,Y -460.475,Z 1016.533,A 0.000,B 0.000,C 90.000,E1 95.910} C_DIS
LIN {X 0.191,Y -449.766,Z 1016.524,A 0.000,B 0.000,C 90.000,E1 94.359} C_DIS
LIN {X -0.124,Y -432.616,Z 1016.510,A 0.000,B 0.000,C 90.000,E1 91.776} C_DIS
LIN {X 0.107,Y -420.145,Z 1016.498,A 0.000,B 0.000,C 90.000,E1 89.599} C_DIS
LIN {X 0.056,Y -408.408,Z 1016.486,A 0.000,B 0.000,C 90.000,E1 87.421} C_DIS
LIN {X 0.067,Y -399.513,Z 1016.476,A 0.000,B 0.000,C 90.000,E1 85.755} C_DIS
LIN {X -0.033,Y -388.841,Z 1016.466,A 0.000,B 0.000,C 90.000,E1 83.799} C_DIS
LIN {X 0.097,Y -379.497,Z 1016.456,A 0.000,B 0.000,C 90.000,E1 82.064} C_DIS
LIN {X 0.055,Y -371.404,Z 1016.448,A 0.000,B 0.000,C 90.000,E1 80.622} C_DIS
LIN {X -0.044,Y -359.854,Z 1016.437,A 0.000,B 0.000,C 90.000,E1 78.578} C_DIS
LIN {X 0.111,Y -349.889,Z 1016.427,A 0.000,B 0.000,C 90.000,E1 76.756} C_DIS
LIN {X -0.151,Y -333.747,Z 1016.410,A 0.000,B 0.000,C 90.000,E1 73.740} C_DIS
LIN {X -0.086,Y -321.342,Z 1016.396,A 0.000,B 0.000,C 90.000,E1 71.221} C_DIS
LIN {X 0.069,Y -310.646,Z 1016.383,A 0.000,B 0.000,C 90.000,E1 68.954} C_DIS
LIN {X -0.008,Y -298.741,Z 1016.369,A 0.000,B 0.000,C 90.000,E1 66.357} C_DIS
LIN {X -0.012,Y -287.116,Z 1016.354,A 0.000,B 0.000,C 90.000,E1 63.691} C_DIS
LIN {X 0.003,Y -277.226,Z 1016.341,A 0.000,B 0.000,C 90.000,E1 61.307} C_DIS
LIN {X 0.066,Y -267.430,Z 1016.327,A 0.000,B 0.000,C 90.000,E1 58.869} C_DIS
LIN {X -0.140,Y -256.478,Z 1016.311,A 0.000,B 0.000,C 90.000,E1 56.087} C_DIS
LIN {X 0.020,Y -244.713,Z 1016.293,A 0.000,B 0.000,C 90.000,E1 52.798} C_DIS
LIN {X 0.055,Y -233.667,Z 1016.275,A 0.000,B 0.000,C 90.000,E1 49.461} C_DIS
LIN {X 0.067,Y -223.278,Z 1016.256,A 0.000,B 0.000,C 90.000,E1 46.053} C_DIS
LIN {X -0.024,Y -215.535,Z 1016.241,A 0.000,B 0.000,C 90.000,E1 43.380} C_DIS
LIN {X -0.043,Y -207.135,Z 1016.224,A 0.000,B 0.000,C 90.000,E1 40.253} C_DIS
LIN {X -0.076,Y -199.311,Z 1016.206,A 0.000,B 0.000,C 90.000,E1 37.076} C_DIS
LIN {X 0.092,Y -192.142,Z 1016.188,A 0.000,B 0.000,C 90.000,E1 33.785} C_DIS
LIN {X -0.068,Y -185.779,Z 1016.170,A 0.000,B 0.000,C 90.000,E1 30.541} C_DIS
LIN {X 0.001,Y -180.269,Z 1016.151,A 0.000,B 0.000,C 90.000,E1 27.180} C_DIS
LIN {X -0.075,Y -175.501,Z 1016.132,A 0.000,B 0.000,C 90.000,E1 23.823} C_DIS
LIN {X 0.016,Y -171.530,Z 1016.113,A 0.000,B 0.000,C 90.000,E1 20.375} C_DIS
LIN {X 0.051,Y -168.199,Z 1016.094,A 0.000,B 0.000,C 90.000,E1 16.913} C_DIS
LIN {X -0.026,Y -165.038,Z 1016.070,A 0.000,B 0.000,C 90.000,E1 12.591} C_DIS
LIN {X 0.082,Y -162.691,Z 1016.041,A 0.000,B 0.000,C 90.000,E1 7.296} C_DIS
LIN {X 0.043,Y -163.608,Z 1015.958,A 0.000,B 0.000,C 90.000,E1 352.470} C_DIS
LIN {X -0.008,Y -166.567,Z 1015.929,A 0.000,B 0.000,C 90.000,E1 347.229} C_DIS
LIN {X -0.092,Y -170.154,Z 1015.905,A 0.000,B 0.000,C 90.000,E1 342.906} C_DIS
LIN {X 0.093,Y -173.864,Z 1015.886,A 0.000,B 0.000,C 90.000,E1 339.390} C_DIS
LIN {X 0.003,Y -178.449,Z 1015.867,A 0.000,B 0.000,C 90.000,E1 335.997} C_DIS
LIN {X -0.010,Y -183.803,Z 1015.848,A 0.000,B 0.000,C 90.000,E1 332.615} C_DIS
LIN {X -0.045,Y -189.964,Z 1015.829,A 0.000,B 0.000,C 90.000,E1 329.282} C_DIS
LIN {X 0.038,Y -196.825,Z 1015.811,A 0.000,B 0.000,C 90.000,E1 325.960} C_DIS
LIN {X 0.027,Y -204.265,Z 1015.793,A 0.000,B 0.000,C 90.000,E1 322.718} C_DIS
LIN {X 0.016,Y -213.364,Z 1015.773,A 0.000,B 0.000,C 90.000,E1 319.138} C_DIS
LIN {X -0.135,Y -221.973,Z 1015.756,A 0.000,B 0.000,C 90.000,E1 316.053} C_DIS
LIN {X 0.079,Y -231.448,Z 1015.739,A 0.000,B 0.000,C 90.000,E1 312.933} C_DIS
LIN {X -0.003,Y -238.134,Z 1015.728,A 0.000,B 0.000,C 90.000,E1 311.067} C_DIS
LIN {X 0.048,Y -245.629,Z 1015.718,A 0.000,B 0.000,C 90.000,E1 309.197} C_DIS
LIN {X -0.074,Y -255.888,Z 1015.706,A 0.000,B 0.000,C 90.000,E1 307.030} C_DIS
LIN {X -0.056,Y -265.425,Z 1015.696,A 0.000,B 0.000,C 90.000,E1 305.231} C_DIS
LIN {X -0.004,Y -282.008,Z 1015.680,A 0.000,B 0.000,C 90.000,E1 302.418} C_DIS
LIN {X 0.056,Y -302.080,Z 1015.663,A 0.000,B 0.000,C 90.000,E1 299.361} C_DIS
LIN {X 0.002,Y -319.110,Z 1015.650,A 0.000,B 0.000,C 90.000,E1 297.078} C_DIS
LIN {X -0.115,Y -332.111,Z 1015.642,A 0.000,B 0.000,C 90.000,E1 295.540} C_DIS
LIN {X -0.134,Y -351.194,Z 1015.630,A 0.000,B 0.000,C 90.000,E1 293.515} C_DIS
LIN {X -0.142,Y -375.924,Z 1015.617,A 0.000,B 0.000,C 90.000,E1 291.153} C_DIS
LIN {X 0.017,Y -389.666,Z 1015.610,A 0.000,B 0.000,C 90.000,E1 289.885} C_DIS
LIN {X -0.099,Y -403.287,Z 1015.604,A 0.000,B 0.000,C 90.000,E1 288.671} C_DIS
LIN {X -0.188,Y -411.193,Z 1015.600,A 0.000,B 0.000,C 90.000,E1 287.946} C_DIS
LIN {X -0.044,Y -418.961,Z 1015.595,A 0.000,B 0.000,C 90.000,E1 287.166} C_DIS
LIN {X -0.083,Y -428.865,Z 1015.590,A 0.000,B 0.000,C 90.000,E1 286.134} C_DIS
LIN {X -0.062,Y -438.394,Z 1015.584,A 0.000,B 0.000,C 90.000,E1 285.064} C_DIS
LIN {X -0.068,Y -447.379,Z 1015.578,A 0.000,B 0.000,C 90.000,E1 284.008} C_DIS
LIN {X -0.131,Y -453.724,Z 1015.573,A 0.000,B 0.000,C 90.000,E1 283.231} C_DIS
LIN {X 0.206,Y -459.569,Z 1015.569,A 0.000,B 0.000,C 90.000,E1 282.411} C_DIS
LIN {X -0.110,Y -466.629,Z 1015.563,A 0.000,B 0.000,C 90.000,E1 281.422} C_DIS
LIN {X -0.114,Y -471.356,Z 1015.559,A 0.000,B 0.000,C 90.000,E1 280.658} C_DIS
LIN {X -0.160,Y -475.508,Z 1015.555,A 0.000,B 0.000,C 90.000,E1 279.905} C_DIS
LIN {X -0.170,Y -479.028,Z 1015.551,A 0.000,B 0.000,C 90.000,E1 279.151} C_DIS
LIN {X 0.051,Y -481.081,Z 1015.548,A 0.000,B 0.000,C 90.000,E1 278.624} C_DIS
LIN {X 0.212,Y -482.799,Z 1015.545,A 0.000,B 0.000,C 90.000,E1 278.106} C_DIS
LIN {X -0.099,Y -484.302,Z 1015.542,A 0.000,B 0.000,C 90.000,E1 277.644} C_DIS
LIN {X -0.211,Y -486.644,Z 1015.537,A 0.000,B 0.000,C 90.000,E1 276.663} C_DIS
LIN {X -0.014,Y -487.492,Z 1015.534,A 0.000,B 0.000,C 90.000,E1 276.144} C_DIS
LIN {X 0.190,Y -488.078,Z 1015.531,A 0.000,B 0.000,C 90.000,E1 275.625} C_DIS
LIN {X -0.087,Y -488.271,Z 1015.529,A 0.000,B 0.000,C 90.000,E1 275.163} C_DIS
LIN {X 0.122,Y -488.047,Z 1015.526,A 0.000,B 0.000,C 90.000,E1 274.645} C_DIS
LIN {X -0.192,Y -487.342,Z 1015.523,A 0.000,B 0.000,C 90.000,E1 274.188} C_DIS
LIN {X 0.015,Y -486.069,Z 1015.520,A 0.000,B 0.000,C 90.000,E1 273.669} C_DIS
LIN {X 0.187,Y -484.276,Z 1015.518,A 0.000,B 0.000,C 90.000,E1 273.154} C_DIS
LIN {X -0.104,Y -481.736,Z 1015.515,A 0.000,B 0.000,C 90.000,E1 272.694} C_DIS
LIN {X 0.046,Y -478.529,Z 1015.512,A 0.000,B 0.000,C 90.000,E1 272.178} C_DIS
LIN {X 0.194,Y -474.473,Z 1015.509,A 0.000,B 0.000,C 90.000,E1 271.661} C_DIS
LIN {X -0.165,Y -469.445,Z 1015.507,A 0.000,B 0.000,C 90.000,E1 271.203} C_DIS
LIN {X 0.112,Y -463.643,Z 1015.504,A 0.000,B 0.000,C 90.000,E1 270.688} C_DIS
LIN {X -0.115,Y -457.339,Z 1015.502,A 0.000,B 0.000,C 90.000,E1 270.286} C_DIS
LIN {X 0.119,Y -450.516,Z 1015.499,A 0.000,B 0.000,C 90.000,E1 269.885} C_DIS
LIN {X -0.023,Y -443.239,Z 1015.498,A 0.000,B 0.000,C 90.000,E1 269.599} C_DIS
LIN {X -0.114,Y -435.691,Z 1015.496,A 0.000,B 0.000,C 90.000,E1 269.370} C_DIS
LIN {X -0.208,Y -427.298,Z 1015.495,A 0.000,B 0.000,C 90.000,E1 269.198} C_DIS
LIN {X 0.122,Y -418.628,Z 1015.495,A 0.000,B 0.000,C 90.000,E1 269.026} C_DIS
LIN {X -0.132,Y -408.641,Z 1015.494,A 0.000,B 0.000,C 90.000,E1 268.969} C_DIS
LIN {X -0.098,Y -397.895,Z 1015.494,A 0.000,B 0.000,C 90.000,E1 268.912} C_DIS
LIN {X -0.073,Y -181.294,Z 1015.494,A 0.000,B 0.000,C 90.000,E1 268.912} C_DIS
LIN {X -0.007,Y -180.893,Z 1015.473,A 0.000,B 0.000,C 90.000,E1 265.179} C_DIS
LIN {X 0.069,Y -179.516,Z 1015.454,A 0.000,B 0.000,C 90.000,E1 261.781} C_DIS
LIN {X 0.055,Y -179.020,Z 1015.445,A 0.000,B 0.000,C 90.000,E1 260.095} C_DIS
LIN {X -0.059,Y -178.653,Z 1015.440,A 0.000,B 0.000,C 90.000,E1 259.285} C_DIS
LIN {X 0.047,Y -175.704,Z 1015.412,A 0.000,B 0.000,C 90.000,E1 254.157} C_DIS
LIN {X 0.057,Y -172.420,Z 1015.388,A 0.000,B 0.000,C 90.000,E1 249.880} C_DIS
LIN {X 0.073,Y -171.240,Z 1015.379,A 0.000,B 0.000,C 90.000,E1 248.156} C_DIS
LIN {X 0.048,Y -167.517,Z 1015.355,A 0.000,B 0.000,C 90.000,E1 243.845} C_DIS
LIN {X -0.019,Y -166.913,Z 1015.350,A 0.000,B 0.000,C 90.000,E1 242.999} C_DIS
LIN {X 0.032,Y -162.221,Z 1015.321,A 0.000,B 0.000,C 90.000,E1 237.740} C_DIS
LIN {X -0.048,Y -160.801,Z 1015.311,A 0.000,B 0.000,C 90.000,E1 236.008} C_DIS
LIN {X -0.068,Y -157.590,Z 1015.291,A 0.000,B 0.000,C 90.000,E1 232.477} C_DIS
LIN {X -0.010,Y -155.623,Z 1015.277,A 0.000,B 0.000,C 90.000,E1 229.784} C_DIS
LIN {X -0.075,Y -151.899,Z 1015.252,A 0.000,B 0.000,C 90.000,E1 225.324} C_DIS
LIN {X -0.060,Y -150.129,Z 1015.237,A 0.000,B 0.000,C 90.000,E1 222.609} C_DIS
LIN {X 0.068,Y -146.918,Z 1015.211,A 0.000,B 0.000,C 90.000,E1 218.016} C_DIS
LIN {X -0.031,Y -145.506,Z 1015.196,A 0.000,B 0.000,C 90.000,E1 215.311} C_DIS
LIN {X -0.035,Y -142.910,Z 1015.171,A 0.000,B 0.000,C 90.000,E1 210.718} C_DIS
LIN {X 0.017,Y -141.530,Z 1015.150,A 0.000,B 0.000,C 90.000,E1 207.001} C_DIS
LIN {X 0.061,Y -139.399,Z 1015.114,A 0.000,B 0.000,C 90.000,E1 200.482} C_DIS
LIN {X -0.020,Y -139.112,Z 1015.104,A 0.000,B 0.000,C 90.000,E1 198.652} C_DIS
LIN {X -0.033,Y -138.353,Z 1015.057,A 0.000,B 0.000,C 90.000,E1 190.254} C_DIS
LIN {X -0.044,Y -139.507,Z 1015.005,A 0.000,B 0.000,C 90.000,E1 180.917} C_DIS
LIN {X 0.038,Y -141.146,Z 1014.974,A 0.000,B 0.000,C 90.000,E1 175.298} C_DIS
LIN {X -0.010,Y -142.527,Z 1014.958,A 0.000,B 0.000,C 90.000,E1 172.534} C_DIS
LIN {X -0.064,Y -144.792,Z 1014.933,A 0.000,B 0.000,C 90.000,E1 167.937} C_DIS
LIN {X 0.065,Y -147.409,Z 1014.912,A 0.000,B 0.000,C 90.000,E1 164.212} C_DIS
LIN {X -0.046,Y -149.985,Z 1014.892,A 0.000,B 0.000,C 90.000,E1 160.604} C_DIS
LIN {X -0.038,Y -153.311,Z 1014.872,A 0.000,B 0.000,C 90.000,E1 156.975} C_DIS
LIN {X 0.014,Y -155.012,Z 1014.862,A 0.000,B 0.000,C 90.000,E1 155.153} C_DIS
LIN {X 0.037,Y -158.656,Z 1014.842,A 0.000,B 0.000,C 90.000,E1 151.563} C_DIS
LIN {X -0.018,Y -161.933,Z 1014.827,A 0.000,B 0.000,C 90.000,E1 148.918} C_DIS
LIN {X 0.005,Y -166.124,Z 1014.808,A 0.000,B 0.000,C 90.000,E1 145.388} C_DIS
LIN {X 0.002,Y -171.134,Z 1014.788,A 0.000,B 0.000,C 90.000,E1 141.904} C_DIS
LIN {X 0.038,Y -176.012,Z 1014.769,A 0.000,B 0.000,C 90.000,E1 138.447} C_DIS
LIN {X 0.034,Y -180.262,Z 1014.755,A 0.000,B 0.000,C 90.000,E1 135.891} C_DIS
LIN {X 0.007,Y -185.676,Z 1014.736,A 0.000,B 0.000,C 90.000,E1 132.528} C_DIS
LIN {X 0.059,Y -190.278,Z 1014.722,A 0.000,B 0.000,C 90.000,E1 130.011} C_DIS
LIN {X 0.099,Y -196.658,Z 1014.702,A 0.000,B 0.000,C 90.000,E1 126.377} C_DIS
LIN {X 0.115,Y -301.391,Z 1014.702,A 0.000,B 0.000,C 90.000,E1 126.377} C_DIS
LIN {X -0.158,Y -303.987,Z 1014.702,A 0.000,B 0.000,C 90.000,E1 126.377} C_DIS
LIN {X -0.030,Y -308.092,Z 1014.701,A 0.000,B 0.000,C 90.000,E1 126.137} C_DIS
LIN {X -0.081,Y -310.530,Z 1014.700,A 0.000,B 0.000,C 90.000,E1 125.931} C_DIS
LIN {X 0.076,Y -314.342,Z 1014.697,A 0.000,B 0.000,C 90.000,E1 125.391} C_DIS
LIN {X -0.135,Y -316.029,Z 1014.695,A 0.000,B 0.000,C 90.000,E1 125.105} C_DIS
LIN {X 0.093,Y -317.352,Z 1014.693,A 0.000,B 0.000,C 90.000,E1 124.739} C_DIS
LIN {X 0.121,Y -328.293,Z 1014.675,A 0.000,B 0.000,C 90.000,E1 121.544} C_DIS
LIN {X 0.021,Y -339.482,Z 1014.660,A 0.000,B 0.000,C 90.000,E1 118.743} C_DIS
LIN {X 0.041,Y -352.080,Z 1014.644,A 0.000,B 0.000,C 90.000,E1 115.976} C_DIS
LIN {X 0.123,Y -366.194,Z 1014.629,A 0.000,B 0.000,C 90.000,E1 113.259} C_DIS
LIN {X 0.054,Y -380.115,Z 1014.616,A 0.000,B 0.000,C 90.000,E1 110.918} C_DIS
LIN {X 0.203,Y -395.435,Z 1014.604,A 0.000,B 0.000,C 90.000,E1 108.598} C_DIS
LIN {X -0.019,Y -412.259,Z 1014.591,A 0.000,B 0.000,C 90.000,E1 106.386} C_DIS
LIN {X 0.062,Y -430.711,Z 1014.579,A 0.000,B 0.000,C 90.000,E1 104.189} C_DIS
LIN {X -0.084,Y -450.550,Z 1014.567,A 0.000,B 0.000,C 90.000,E1 102.119} C_DIS
LIN {X -0.039,Y -468.245,Z 1014.558,A 0.000,B 0.000,C 90.000,E1 100.423} C_DIS
LIN {X -0.190,Y -470.139,Z 1014.557,A 0.000,B 0.000,C 90.000,E1 100.197} C_DIS
LIN {X 0.206,Y -471.575,Z 1014.555,A 0.000,B 0.000,C 90.000,E1 99.905} C_DIS
LIN {X -0.085,Y -473.504,Z 1014.552,A 0.000,B 0.000,C 90.000,E1 99.434} C_DIS
LIN {X 0.022,Y -474.320,Z 1014.550,A 0.000,B 0.000,C 90.000,E1 98.916} C_DIS
LIN {X 0.142,Y -474.162,Z 1014.547,A 0.000,B 0.000,C 90.000,E1 98.398} C_DIS
LIN {X -0.200,Y -473.013,Z 1014.544,A 0.000,B 0.000,C 90.000,E1 97.936} C_DIS
LIN {X 0.130,Y -472.014,Z 1014.543,A 0.000,B 0.000,C 90.000,E1 97.644} C_DIS
LIN {X -0.010,Y -470.670,Z 1014.541,A 0.000,B 0.000,C 90.000,E1 97.409} C_DIS
LIN {X -0.191,Y -460.220,Z 1014.533,A 0.000,B 0.000,C 90.000,E1 95.910} C_DIS
LIN {X -0.129,Y -449.517,Z 1014.524,A 0.000,B 0.000,C 90.000,E1 94.359} C_DIS
LIN {X 0.143,Y -430.771,Z 1014.508,A 0.000,B 0.000,C 90.000,E1 91.432} C_DIS
LIN {X 0.118,Y -415.505,Z 1014.493,A 0.000,B 0.000,C 90.000,E1 88.740} C_DIS
LIN {X -0.086,Y -405.262,Z 1014.482,A 0.000,B 0.000,C 90.000,E1 86.846} C_DIS
LIN {X -0.123,Y -396.251,Z 1014.473,A 0.000,B 0.000,C 90.000,E1 85.179} C_DIS
LIN {X 0.059,Y -387.090,Z 1014.464,A 0.000,B 0.000,C 90.000,E1 83.457} C_DIS
LIN {X 0.147,Y -377.690,Z 1014.454,A 0.000,B 0.000,C 90.000,E1 81.724} C_DIS
LIN {X 0.124,Y -369.524,Z 1014.446,A 0.000,B 0.000,C 90.000,E1 80.274} C_DIS
LIN {X -0.011,Y -357.957,Z 1014.435,A 0.000,B 0.000,C 90.000,E1 78.229} C_DIS
LIN {X -0.040,Y -344.715,Z 1014.421,A 0.000,B 0.000,C 90.000,E1 75.825} C_DIS
LIN {X 0.067,Y -330.408,Z 1014.406,A 0.000,B 0.000,C 90.000,E1 73.032} C_DIS
LIN {X -0.164,Y -318.054,Z 1014.392,A 0.000,B 0.000,C 90.000,E1 70.550} C_DIS
LIN {X 0.117,Y -305.930,Z 1014.377,A 0.000,B 0.000,C 90.000,E1 67.922} C_DIS
LIN {X 0.032,Y -294.133,Z 1014.363,A 0.000,B 0.000,C 90.000,E1 65.305} C_DIS
LIN {X 0.032,Y -282.684,Z 1014.348,A 0.000,B 0.000,C 90.000,E1 62.615} C_DIS
LIN {X 0.077,Y -272.807,Z 1014.335,A 0.000,B 0.000,C 90.000,E1 60.205} C_DIS
LIN {X -0.141,Y -261.691,Z 1014.319,A 0.000,B 0.000,C 90.000,E1 57.454} C_DIS
LIN {X 0.028,Y -249.665,Z 1014.301,A 0.000,B 0.000,C 90.000,E1 54.196} C_DIS
LIN {X 0.094,Y -238.257,Z 1014.283,A 0.000,B 0.000,C 90.000,E1 50.884} C_DIS
LIN {X -0.075,Y -227.601,Z 1014.264,A 0.000,B 0.000,C 90.000,E1 47.553} C_DIS
LIN {X -0.076,Y -217.504,Z 1014.245,A 0.000,B 0.000,C 90.000,E1 44.109} C_DIS
LIN {X -0.068,Y -208.974,Z 1014.228,A 0.000,B 0.000,C 90.000,E1 40.987} C_DIS
LIN {X -0.057,Y -200.973,Z 1014.210,A 0.000,B 0.000,C 90.000,E1 37.810} C_DIS
LIN {X -0.004,Y -193.639,Z 1014.192,A 0.000,B 0.000,C 90.000,E1 34.565} C_DIS
LIN {X 0.076,Y -187.100,Z 1014.174,A 0.000,B 0.000,C 90.000,E1 31.258} C_DIS
LIN {X -0.073,Y -181.410,Z 1014.155,A 0.000,B 0.000,C 90.000,E1 27.975} C_DIS
LIN {X -0.037,Y -176.477,Z 1014.137,A 0.000,B 0.000,C 90.000,E1 24.591} C_DIS
LIN {X 0.047,Y -172.331,Z 1014.118,A 0.000,B 0.000,C 90.000,E1 21.153} C_DIS
LIN {X 0.096,Y -168.867,Z 1014.098,A 0.000,B 0.000,C 90.000,E1 17.692} C_DIS
LIN {X 0.079,Y -165.503,Z 1014.074,A 0.000,B 0.000,C 90.000,E1 13.355} C_DIS
LIN {X 0.069,Y -162.908,Z 1014.045,A 0.000,B 0.000,C 90.000,E1 8.106} C_DIS
LIN {X 0.042,Y -163.574,Z 1013.958,A 0.000,B 0.000,C 90.000,E1 352.470} C_DIS
LIN {X -0.011,Y -166.521,Z 1013.929,A 0.000,B 0.000,C 90.000,E1 347.229} C_DIS
LIN {X -0.097,Y -170.120,Z 1013.905,A 0.000,B 0.000,C 90.000,E1 342.906} C_DIS
LIN {X 0.088,Y -173.844,Z 1013.886,A 0.000,B 0.000,C 90.000,E1 339.390} C_DIS
LIN {X -0.002,Y -178.451,Z 1013.867,A 0.000,B 0.000,C 90.000,E1 335.997} C_DIS
LIN {X -0.015,Y -183.816,Z 1013.848,A 0.000,B 0.000,C 90.000,E1 332.615} C_DIS
LIN {X -0.050,Y -189.990,Z 1013.829,A 0.000,B 0.000,C 90.000,E1 329.282} C_DIS
LIN {X 0.034,Y -196.860,Z 1013.811,A 0.000,B 0.000,C 90.000,E1 325.960} C_DIS
LIN {X 0.023,Y -204.279,Z 1013.793,A 0.000,B 0.000,C 90.000,E1 322.718} C_DIS
LIN {X 0.012,Y -213.391,Z 1013.773,A 0.000,B 0.000,C 90.000,E1 319.138} C_DIS
LIN {X -0.139,Y -221.971,Z 1013.756,A 0.000,B 0.000,C 90.000,E1 316.053} C_DIS
LIN {X 0.075,Y -231.422,Z 1013.739,A 0.000,B 0.000,C 90.000,E1 312.933} C_DIS
LIN {X -0.007,Y -238.112,Z 1013.728,A 0.000,B 0.000,C 90.000,E1 311.067} C_DIS
LIN {X 0.042,Y -245.631,Z 1013.718,A 0.000,B 0.000,C 90.000,E1 309.197} C_DIS
LIN {X 0.075,Y -255.904,Z 1013.706,A 0.000,B 0.000,C 90.000,E1 306.996} C_DIS
LIN {X -0.007,Y -267.461,Z 1013.694,A 0.000,B 0.000,C 90.000,E1 304.865} C_DIS
LIN {X -0.008,Y -282.061,Z 1013.680,A 0.000,B 0.000,C 90.000,E1 302.418} C_DIS
LIN {X 0.053,Y -302.144,Z 1013.663,A 0.000,B 0.000,C 90.000,E1 299.361} C_DIS
LIN {X 0.000,Y -319.196,Z 1013.650,A 0.000,B 0.000,C 90.000,E1 297.078} C_DIS
LIN {X -0.128,Y -332.238,Z 1013.642,A 0.000,B 0.000,C 90.000,E1 295.540} C_DIS
LIN {X -0.001,Y -353.686,Z 1013.629,A 0.000,B 0.000,C 90.000,E1 293.259} C_DIS
LIN {X -0.061,Y -378.472,Z 1013.616,A 0.000,B 0.000,C 90.000,E1 290.918} C_DIS
LIN {X -0.136,Y -392.197,Z 1013.609,A 0.000,B 0.000,C 90.000,E1 289.685} C_DIS
LIN {X 0.114,Y -405.751,Z 1013.602,A 0.000,B 0.000,C 90.000,E1 288.417} C_DIS
LIN {X -0.025,Y -413.602,Z 1013.598,A 0.000,B 0.000,C 90.000,E1 287.692} C_DIS
LIN {X 0.063,Y -421.245,Z 1013.594,A 0.000,B 0.000,C 90.000,E1 286.913} C_DIS
LIN {X -0.159,Y -431.040,Z 1013.588,A 0.000,B 0.000,C 90.000,E1 285.898} C_DIS
LIN {X 0.071,Y -438.180,Z 1013.584,A 0.000,B 0.000,C 90.000,E1 285.064} C_DIS
LIN {X 0.045,Y -447.156,Z 1013.578,A 0.000,B 0.000,C 90.000,E1 284.008} C_DIS
LIN {X 0.133,Y -455.532,Z 1013.572,A 0.000,B 0.000,C 90.000,E1 282.952} C_DIS
LIN {X 0.040,Y -461.250,Z 1013.568,A 0.000,B 0.000,C 90.000,E1 282.187} C_DIS
LIN {X 0.000,Y -466.467,Z 1013.563,A 0.000,B 0.000,C 90.000,E1 281.422} C_DIS
LIN {X -0.149,Y -472.725,Z 1013.558,A 0.000,B 0.000,C 90.000,E1 280.423} C_DIS
LIN {X -0.188,Y -476.698,Z 1013.554,A 0.000,B 0.000,C 90.000,E1 279.670} C_DIS
LIN {X -0.059,Y -479.011,Z 1013.551,A 0.000,B 0.000,C 90.000,E1 279.151} C_DIS
LIN {X 0.161,Y -481.051,Z 1013.548,A 0.000,B 0.000,C 90.000,E1 278.624} C_DIS
LIN {X -0.163,Y -482.837,Z 1013.545,A 0.000,B 0.000,C 90.000,E1 278.163} C_DIS
LIN {X 0.006,Y -484.344,Z 1013.542,A 0.000,B 0.000,C 90.000,E1 277.644} C_DIS
LIN {X 0.187,Y -485.621,Z 1013.540,A 0.000,B 0.000,C 90.000,E1 277.125} C_DIS
LIN {X -0.106,Y -486.718,Z 1013.537,A 0.000,B 0.000,C 90.000,E1 276.663} C_DIS
LIN {X 0.092,Y -487.577,Z 1013.534,A 0.000,B 0.000,C 90.000,E1 276.144} C_DIS
LIN {X -0.189,Y -488.186,Z 1013.531,A 0.000,B 0.000,C 90.000,E1 275.682} C_DIS
LIN {X 0.019,Y -488.397,Z 1013.529,A 0.000,B 0.000,C 90.000,E1 275.163} C_DIS
LIN {X 0.230,Y -488.179,Z 1013.526,A 0.000,B 0.000,C 90.000,E1 274.645} C_DIS
LIN {X -0.084,Y -487.507,Z 1013.523,A 0.000,B 0.000,C 90.000,E1 274.188} C_DIS
LIN {X 0.124,Y -486.311,Z 1013.520,A 0.000,B 0.000,C 90.000,E1 273.669} C_DIS
LIN {X -0.187,Y -484.518,Z 1013.518,A 0.000,B 0.000,C 90.000,E1 273.212} C_DIS
LIN {X 0.006,Y -482.071,Z 1013.515,A 0.000,B 0.000,C 90.000,E1 272.694} C_DIS
LIN {X -0.159,Y -480.569,Z 1013.514,A 0.000,B 0.000,C 90.000,E1 272.465} C_DIS
LIN {X -0.014,Y -476.964,Z 1013.511,A 0.000,B 0.000,C 90.000,E1 271.949} C_DIS
LIN {X 0.126,Y -472.509,Z 1013.508,A 0.000,B 0.000,C 90.000,E1 271.432} C_DIS
LIN {X -0.140,Y -467.137,Z 1013.505,A 0.000,B 0.000,C 90.000,E1 270.974} C_DIS
LIN {X -0.096,Y -461.223,Z 1013.503,A 0.000,B 0.000,C 90.000,E1 270.516} C_DIS
LIN {X -0.061,Y -454.850,Z 1013.501,A 0.000,B 0.000,C 90.000,E1 270.115} C_DIS
LIN {X -0.006,Y -448.002,Z 1013.499,A 0.000,B 0.000,C 90.000,E1 269.771} C_DIS
LIN {X 0.083,Y -440.760,Z 1013.497,A 0.000,B 0.000,C 90.000,E1 269.484} C_DIS
LIN {X 0.171,Y -433.078,Z 1013.496,A 0.000,B 0.000,C 90.000,E1 269.255} C_DIS
LIN {X -0.203,Y -424.752,Z 1013.495,A 0.000,B 0.000,C 90.000,E1 269.141} C_DIS
LIN {X 0.202,Y -415.664,Z 1013.494,A 0.000,B 0.000,C 90.000,E1 268.969} C_DIS
LIN {X -0.123,Y -401.058,Z 1013.494,A 0.000,B 0.000,C 90.000,E1 268.912} C_DIS
LIN {X -0.185,Y -398.544,Z 1013.494,A 0.000,B 0.000,C 90.000,E1 268.912} C_DIS
LIN {X 0.068,Y -181.291,Z 1013.494,A 0.000,B 0.000,C 90.000,E1 268.854} C_DIS
LIN {X -0.047,Y -180.891,Z 1013.473,A 0.000,B 0.000,C 90.000,E1 265.179} C_DIS
LIN {X 0.015,Y -179.017,Z 1013.445,A 0.000,B 0.000,C 90.000,E1 260.095} C_DIS
LIN {X -0.066,Y -178.644,Z 1013.440,A 0.000,B 0.000,C 90.000,E1 259.275} C_DIS
LIN {X 0.008,Y -175.695,Z 1013.412,A 0.000,B 0.000,C 90.000,E1 254.157} C_DIS
LIN {X 0.018,Y -172.412,Z 1013.388,A 0.000,B 0.000,C 90.000,E1 249.880} C_DIS
LIN {X 0.035,Y -171.227,Z 1013.379,A 0.000,B 0.000,C 90.000,E1 248.156} C_DIS
LIN {X 0.010,Y -167.508,Z 1013.355,A 0.000,B 0.000,C 90.000,E1 243.845} C_DIS
LIN {X -0.057,Y -166.903,Z 1013.350,A 0.000,B 0.000,C 90.000,E1 242.999} C_DIS
LIN {X -0.005,Y -162.211,Z 1013.321,A 0.000,B 0.000,C 90.000,E1 237.740} C_DIS
LIN {X 0.048,Y -160.788,Z 1013.311,A 0.000,B 0.000,C 90.000,E1 235.960} C_DIS
LIN {X 0.020,Y -157.579,Z 1013.291,A 0.000,B 0.000,C 90.000,E1 232.431} C_DIS
LIN {X 0.053,Y -155.611,Z 1013.276,A 0.000,B 0.000,C 90.000,E1 229.747} C_DIS
LIN {X -0.003,Y -151.890,Z 1013.252,A 0.000,B 0.000,C 90.000,E1 225.283} C_DIS
LIN {X -0.096,Y -150.118,Z 1013.237,A 0.000,B 0.000,C 90.000,E1 222.609} C_DIS
LIN {X 0.033,Y -146.911,Z 1013.211,A 0.000,B 0.000,C 90.000,E1 218.016} C_DIS
LIN {X -0.066,Y -145.498,Z 1013.196,A 0.000,B 0.000,C 90.000,E1 215.311} C_DIS
LIN {X 0.053,Y -142.903,Z 1013.170,A 0.000,B 0.000,C 90.000,E1 210.669} C_DIS
LIN {X -0.017,Y -141.523,Z 1013.150,A 0.000,B 0.000,C 90.000,E1 207.001} C_DIS
LIN {X 0.027,Y -139.396,Z 1013.114,A 0.000,B 0.000,C 90.000,E1 200.482} C_DIS
LIN {X 0.077,Y -139.108,Z 1013.104,A 0.000,B 0.000,C 90.000,E1 198.598} C_DIS
LIN {X -0.068,Y -138.353,Z 1013.057,A 0.000,B 0.000,C 90.000,E1 190.254} C_DIS
LIN {X 0.062,Y -139.510,Z 1013.005,A 0.000,B 0.000,C 90.000,E1 180.859} C_DIS
LIN {X 0.003,Y -141.152,Z 1012.974,A 0.000,B 0.000,C 90.000,E1 175.298} C_DIS
LIN {X -0.026,Y -142.532,Z 1012.958,A 0.000,B 0.000,C 90.000,E1 172.527} C_DIS
LIN {X 0.042,Y -144.800,Z 1012.933,A 0.000,B 0.000,C 90.000,E1 167.881} C_DIS
LIN {X 0.031,Y -147.419,Z 1012.912,A 0.000,B 0.000,C 90.000,E1 164.212} C_DIS
LIN {X 0.060,Y -149.996,Z 1012.892,A 0.000,B 0.000,C 90.000,E1 160.550} C_DIS
LIN {X 0.067,Y -153.324,Z 1012.872,A 0.000,B 0.000,C 90.000,E1 156.922} C_DIS
LIN {X -0.022,Y -155.025,Z 1012.862,A 0.000,B 0.000,C 90.000,E1 155.153} C_DIS
LIN {X 0.000,Y -158.671,Z 1012.842,A 0.000,B 0.000,C 90.000,E1 151.563} C_DIS
LIN {X 0.083,Y -161.950,Z 1012.827,A 0.000,B 0.000,C 90.000,E1 148.869} C_DIS
LIN {X -0.032,Y -166.141,Z 1012.808,A 0.000,B 0.000,C 90.000,E1 145.388} C_DIS
LIN {X -0.036,Y -171.153,Z 1012.788,A 0.000,B 0.000,C 90.000,E1 141.904} C_DIS
LIN {X -0.002,Y -176.032,Z 1012.769,A 0.000,B 0.000,C 90.000,E1 138.447} C_DIS
LIN {X -0.007,Y -180.285,Z 1012.755,A 0.000,B 0.000,C 90.000,E1 135.891} C_DIS
LIN {X -0.034,Y -185.697,Z 1012.736,A 0.000,B 0.000,C 90.000,E1 132.528} C_DIS
LIN {X 0.018,Y -190.302,Z 1012.722,A 0.000,B 0.000,C 90.000,E1 130.011} C_DIS
LIN {X -0.047,Y -196.587,Z 1012.702,A 0.000,B 0.000,C 90.000,E1 126.457} C_DIS
LIN {X 0.071,Y -301.529,Z 1012.702,A 0.000,B 0.000,C 90.000,E1 126.423} C_DIS
LIN {X 0.089,Y -303.627,Z 1012.702,A 0.000,B 0.000,C 90.000,E1 126.377} C_DIS
LIN {X -0.118,Y -308.243,Z 1012.701,A 0.000,B 0.000,C 90.000,E1 126.171} C_DIS
LIN {X 0.105,Y -310.867,Z 1012.699,A 0.000,B 0.000,C 90.000,E1 125.884} C_DIS
LIN {X -0.117,Y -314.620,Z 1012.696,A 0.000,B 0.000,C 90.000,E1 125.391} C_DIS
LIN {X 0.112,Y -316.214,Z 1012.695,A 0.000,B 0.000,C 90.000,E1 125.025} C_DIS
LIN {X -0.034,Y -318.500,Z 1012.691,A 0.000,B 0.000,C 90.000,E1 124.405} C_DIS
LIN {X 0.033,Y -329.576,Z 1012.673,A 0.000,B 0.000,C 90.000,E1 121.209} C_DIS
LIN {X -0.039,Y -340.935,Z 1012.658,A 0.000,B 0.000,C 90.000,E1 118.409} C_DIS
LIN {X -0.133,Y -353.710,Z 1012.642,A 0.000,B 0.000,C 90.000,E1 115.668} C_DIS
LIN {X -0.085,Y -366.351,Z 1012.629,A 0.000,B 0.000,C 90.000,E1 113.259} C_DIS
LIN {X -0.158,Y -380.291,Z 1012.616,A 0.000,B 0.000,C 90.000,E1 110.918} C_DIS
LIN {X -0.012,Y -395.629,Z 1012.603,A 0.000,B 0.000,C 90.000,E1 108.598} C_DIS
LIN {X -0.123,Y -412.476,Z 1012.591,A 0.000,B 0.000,C 90.000,E1 106.370} C_DIS
LIN {X -0.056,Y -430.950,Z 1012.579,A 0.000,B 0.000,C 90.000,E1 104.175} C_DIS
LIN {X 0.140,Y -450.799,Z 1012.567,A 0.000,B 0.000,C 90.000,E1 102.063} C_DIS
LIN {X 0.201,Y -466.087,Z 1012.559,A 0.000,B 0.000,C 90.000,E1 100.602} C_DIS
LIN {X 0.211,Y -468.446,Z 1012.558,A 0.000,B 0.000,C 90.000,E1 100.366} C_DIS
LIN {X 0.035,Y -470.308,Z 1012.556,A 0.000,B 0.000,C 90.000,E1 100.141} C_DIS
LIN {X -0.058,Y -471.717,Z 1012.555,A 0.000,B 0.000,C 90.000,E1 99.905} C_DIS
LIN {X 0.119,Y -473.572,Z 1012.552,A 0.000,B 0.000,C 90.000,E1 99.378} C_DIS
LIN {X 0.226,Y -474.327,Z 1012.549,A 0.000,B 0.000,C 90.000,E1 98.859} C_DIS
LIN {X -0.121,Y -474.112,Z 1012.547,A 0.000,B 0.000,C 90.000,E1 98.398} C_DIS
LIN {X 0.072,Y -472.901,Z 1012.544,A 0.000,B 0.000,C 90.000,E1 97.871} C_DIS
LIN {X -0.132,Y -471.864,Z 1012.542,A 0.000,B 0.000,C 90.000,E1 97.644} C_DIS
LIN {X 0.195,Y -470.473,Z 1012.541,A 0.000,B 0.000,C 90.000,E1 97.352} C_DIS
LIN {X 0.009,Y -460.014,Z 1012.533,A 0.000,B 0.000,C 90.000,E1 95.853} C_DIS
LIN {X 0.063,Y -449.324,Z 1012.524,A 0.000,B 0.000,C 90.000,E1 94.302} C_DIS
LIN {X -0.108,Y -430.610,Z 1012.508,A 0.000,B 0.000,C 90.000,E1 91.432} C_DIS
LIN {X -0.130,Y -415.350,Z 1012.493,A 0.000,B 0.000,C 90.000,E1 88.740} C_DIS
LIN {X 0.075,Y -405.110,Z 1012.482,A 0.000,B 0.000,C 90.000,E1 86.788} C_DIS
LIN {X 0.031,Y -396.078,Z 1012.473,A 0.000,B 0.000,C 90.000,E1 85.122} C_DIS
LIN {X -0.136,Y -386.916,Z 1012.464,A 0.000,B 0.000,C 90.000,E1 83.451} C_DIS
LIN {X -0.089,Y -377.492,Z 1012.454,A 0.000,B 0.000,C 90.000,E1 81.724} C_DIS
LIN {X -0.110,Y -369.341,Z 1012.446,A 0.000,B 0.000,C 90.000,E1 80.274} C_DIS
LIN {X 0.109,Y -357.761,Z 1012.434,A 0.000,B 0.000,C 90.000,E1 78.173} C_DIS
LIN {X 0.152,Y -344.531,Z 1012.421,A 0.000,B 0.000,C 90.000,E1 75.755} C_DIS
LIN {X -0.058,Y -330.232,Z 1012.406,A 0.000,B 0.000,C 90.000,E1 73.015} C_DIS
LIN {X 0.083,Y -319.410,Z 1012.393,A 0.000,B 0.000,C 90.000,E1 70.786} C_DIS
LIN {X -0.005,Y -307.267,Z 1012.379,A 0.000,B 0.000,C 90.000,E1 68.230} C_DIS
LIN {X -0.051,Y -295.439,Z 1012.364,A 0.000,B 0.000,C 90.000,E1 65.613} C_DIS
LIN {X -0.012,Y -283.944,Z 1012.350,A 0.000,B 0.000,C 90.000,E1 62.922} C_DIS
LIN {X -0.069,Y -274.053,Z 1012.336,A 0.000,B 0.000,C 90.000,E1 60.539} C_DIS
LIN {X -0.032,Y -262.889,Z 1012.321,A 0.000,B 0.000,C 90.000,E1 57.740} C_DIS
LIN {X -0.037,Y -250.795,Z 1012.303,A 0.000,B 0.000,C 90.000,E1 54.529} C_DIS
LIN {X -0.083,Y -239.311,Z 1012.285,A 0.000,B 0.000,C 90.000,E1 51.251} C_DIS
LIN {X -0.040,Y -228.554,Z 1012.266,A 0.000,B 0.000,C 90.000,E1 47.877} C_DIS
LIN {X -0.095,Y -219.515,Z 1012.249,A 0.000,B 0.000,C 90.000,E1 44.838} C_DIS
LIN {X 0.100,Y -210.840,Z 1012.232,A 0.000,B 0.000,C 90.000,E1 41.676} C_DIS
LIN {X -0.006,Y -202.722,Z 1012.214,A 0.000,B 0.000,C 90.000,E1 38.543} C_DIS
LIN {X 0.045,Y -195.220,Z 1012.196,A 0.000,B 0.000,C 90.000,E1 35.311} C_DIS
LIN {X -0.001,Y -188.494,Z 1012.178,A 0.000,B 0.000,C 90.000,E1 32.054} C_DIS
LIN {X -0.029,Y -182.623,Z 1012.160,A 0.000,B 0.000,C 90.000,E1 28.743} C_DIS
LIN {X 0.109,Y -177.530,Z 1012.141,A 0.000,B 0.000,C 90.000,E1 25.335} C_DIS
LIN {X -0.012,Y -173.190,Z 1012.122,A 0.000,B 0.000,C 90.000,E1 21.972} C_DIS
LIN {X -0.037,Y -169.582,Z 1012.103,A 0.000,B 0.000,C 90.000,E1 18.544} C_DIS
LIN {X 0.020,Y -166.009,Z 1012.079,A 0.000,B 0.000,C 90.000,E1 14.189} C_DIS
LIN {X -0.066,Y -163.184,Z 1012.050,A 0.000,B 0.000,C 90.000,E1 8.973} C_DIS
LIN {X 0.007,Y -163.939,Z 1011.953,A 0.000,B 0.000,C 90.000,E1 351.602} C_DIS
LIN {X -0.014,Y -166.487,Z 1011.929,A 0.000,B 0.000,C 90.000,E1 347.229} C_DIS
LIN {X 0.062,Y -170.094,Z 1011.905,A 0.000,B 0.000,C 90.000,E1 342.851} C_DIS
LIN {X 0.083,Y -173.837,Z 1011.886,A 0.000,B 0.000,C 90.000,E1 339.390} C_DIS
LIN {X -0.007,Y -178.452,Z 1011.867,A 0.000,B 0.000,C 90.000,E1 335.997} C_DIS
LIN {X -0.020,Y -183.836,Z 1011.848,A 0.000,B 0.000,C 90.000,E1 332.615} C_DIS
LIN {X -0.054,Y -190.032,Z 1011.829,A 0.000,B 0.000,C 90.000,E1 329.282} C_DIS
LIN {X 0.030,Y -196.893,Z 1011.811,A 0.000,B 0.000,C 90.000,E1 325.960} C_DIS
LIN {X 0.020,Y -204.302,Z 1011.793,A 0.000,B 0.000,C 90.000,E1 322.718} C_DIS
LIN {X 0.010,Y -213.417,Z 1011.773,A 0.000,B 0.000,C 90.000,E1 319.138} C_DIS
LIN {X -0.141,Y -221.975,Z 1011.756,A 0.000,B 0.000,C 90.000,E1 316.053} C_DIS
LIN {X 0.073,Y -231.383,Z 1011.739,A 0.000,B 0.000,C 90.000,E1 312.933} C_DIS
LIN {X -0.011,Y -238.071,Z 1011.728,A 0.000,B 0.000,C 90.000,E1 311.067} C_DIS
LIN {X 0.039,Y -245.634,Z 1011.718,A 0.000,B 0.000,C 90.000,E1 309.197} C_DIS
LIN {X 0.072,Y -255.922,Z 1011.706,A 0.000,B 0.000,C 90.000,E1 306.996} C_DIS
LIN {X -0.109,Y -269.531,Z 1011.692,A 0.000,B 0.000,C 90.000,E1 304.532} C_DIS
LIN {X 0.048,Y -286.469,Z 1011.676,A 0.000,B 0.000,C 90.000,E1 301.720} C_DIS
LIN {X 0.087,Y -306.970,Z 1011.659,A 0.000,B 0.000,C 90.000,E1 298.693} C_DIS
LIN {X 0.002,Y -319.284,Z 1011.650,A 0.000,B 0.000,C 90.000,E1 297.078} C_DIS
LIN {X -0.137,Y -332.361,Z 1011.642,A 0.000,B 0.000,C 90.000,E1 295.540} C_DIS
LIN {X 0.001,Y -353.798,Z 1011.629,A 0.000,B 0.000,C 90.000,E1 293.259} C_DIS
LIN {X 0.078,Y -375.787,Z 1011.618,A 0.000,B 0.000,C 90.000,E1 291.153} C_DIS
LIN {X 0.205,Y -392.336,Z 1011.609,A 0.000,B 0.000,C 90.000,E1 289.631} C_DIS
LIN {X 0.055,Y -403.079,Z 1011.604,A 0.000,B 0.000,C 90.000,E1 288.671} C_DIS
LIN {X -0.004,Y -413.526,Z 1011.598,A 0.000,B 0.000,C 90.000,E1 287.692} C_DIS
LIN {X 0.093,Y -421.146,Z 1011.594,A 0.000,B 0.000,C 90.000,E1 286.913} C_DIS
LIN {X -0.179,Y -430.992,Z 1011.588,A 0.000,B 0.000,C 90.000,E1 285.898} C_DIS
LIN {X -0.186,Y -440.397,Z 1011.582,A 0.000,B 0.000,C 90.000,E1 284.828} C_DIS
LIN {X -0.188,Y -449.257,Z 1011.576,A 0.000,B 0.000,C 90.000,E1 283.772} C_DIS
LIN {X 0.022,Y -457.422,Z 1011.571,A 0.000,B 0.000,C 90.000,E1 282.703} C_DIS
LIN {X 0.133,Y -464.739,Z 1011.565,A 0.000,B 0.000,C 90.000,E1 281.658} C_DIS
LIN {X 0.123,Y -469.669,Z 1011.561,A 0.000,B 0.000,C 90.000,E1 280.894} C_DIS
LIN {X 0.061,Y -474.119,Z 1011.556,A 0.000,B 0.000,C 90.000,E1 280.141} C_DIS
LIN {X 0.123,Y -477.921,Z 1011.552,A 0.000,B 0.000,C 90.000,E1 279.378} C_DIS
LIN {X 0.134,Y -481.111,Z 1011.548,A 0.000,B 0.000,C 90.000,E1 278.624} C_DIS
LIN {X -0.183,Y -482.908,Z 1011.545,A 0.000,B 0.000,C 90.000,E1 278.163} C_DIS
LIN {X -0.014,Y -484.425,Z 1011.542,A 0.000,B 0.000,C 90.000,E1 277.644} C_DIS
LIN {X 0.167,Y -485.739,Z 1011.540,A 0.000,B 0.000,C 90.000,E1 277.125} C_DIS
LIN {X -0.125,Y -486.812,Z 1011.537,A 0.000,B 0.000,C 90.000,E1 276.663} C_DIS
LIN {X 0.074,Y -487.673,Z 1011.534,A 0.000,B 0.000,C 90.000,E1 276.144} C_DIS
LIN {X -0.207,Y -488.294,Z 1011.531,A 0.000,B 0.000,C 90.000,E1 275.682} C_DIS
LIN {X 0.002,Y -488.522,Z 1011.529,A 0.000,B 0.000,C 90.000,E1 275.163} C_DIS
LIN {X 0.212,Y -488.368,Z 1011.526,A 0.000,B 0.000,C 90.000,E1 274.645} C_DIS
LIN {X -0.100,Y -487.693,Z 1011.523,A 0.000,B 0.000,C 90.000,E1 274.188} C_DIS
LIN {X 0.110,Y -486.519,Z 1011.520,A 0.000,B 0.000,C 90.000,E1 273.669} C_DIS
LIN {X -0.201,Y -484.733,Z 1011.518,A 0.000,B 0.000,C 90.000,E1 273.212} C_DIS
LIN {X -0.007,Y -482.290,Z 1011.515,A 0.000,B 0.000,C 90.000,E1 272.694} C_DIS
LIN {X -0.171,Y -480.814,Z 1011.514,A 0.000,B 0.000,C 90.000,E1 272.465} C_DIS
LIN {X -0.024,Y -477.189,Z 1011.511,A 0.000,B 0.000,C 90.000,E1 271.949} C_DIS
LIN {X 0.116,Y -472.740,Z 1011.508,A 0.000,B 0.000,C 90.000,E1 271.432} C_DIS
LIN {X -0.167,Y -467.402,Z 1011.505,A 0.000,B 0.000,C 90.000,E1 270.974} C_DIS
LIN {X -0.119,Y -461.461,Z 1011.503,A 0.000,B 0.000,C 90.000,E1 270.516} C_DIS
LIN {X -0.064,Y -455.160,Z 1011.501,A 0.000,B 0.000,C 90.000,E1 270.115} C_DIS
LIN {X -0.004,Y -448.380,Z 1011.499,A 0.000,B 0.000,C 90.000,E1 269.771} C_DIS
LIN {X 0.088,Y -441.173,Z 1011.497,A 0.000,B 0.000,C 90.000,E1 269.484} C_DIS
LIN {X 0.162,Y -433.558,Z 1011.496,A 0.000,B 0.000,C 90.000,E1 269.255} C_DIS
LIN {X 0.173,Y -425.185,Z 1011.495,A 0.000,B 0.000,C 90.000,E1 269.083} C_DIS
LIN {X 0.120,Y -416.075,Z 1011.494,A 0.000,B 0.000,C 90.000,E1 268.969} C_DIS
LIN {X 0.187,Y -401.621,Z 1011.494,A 0.000,B 0.000,C 90.000,E1 268.854} C_DIS
LIN {X 0.122,Y -399.065,Z 1011.494,A 0.000,B 0.000,C 90.000,E1 268.854} C_DIS
LIN {X 0.026,Y -181.288,Z 1011.494,A 0.000,B 0.000,C 90.000,E1 268.854} C_DIS
LIN {X 0.090,Y -180.890,Z 1011.473,A 0.000,B 0.000,C 90.000,E1 265.122} C_DIS
LIN {X -0.028,Y -179.013,Z 1011.445,A 0.000,B 0.000,C 90.000,E1 260.095} C_DIS
LIN {X 0.067,Y -178.635,Z 1011.440,A 0.000,B 0.000,C 90.000,E1 259.218} C_DIS
LIN {X -0.035,Y -175.686,Z 1011.412,A 0.000,B 0.000,C 90.000,E1 254.157} C_DIS
LIN {X -0.024,Y -172.402,Z 1011.388,A 0.000,B 0.000,C 90.000,E1 249.880} C_DIS
LIN {X -0.008,Y -171.213,Z 1011.379,A 0.000,B 0.000,C 90.000,E1 248.156} C_DIS
LIN {X -0.030,Y -167.498,Z 1011.355,A 0.000,B 0.000,C 90.000,E1 243.845} C_DIS
LIN {X 0.051,Y -166.894,Z 1011.350,A 0.000,B 0.000,C 90.000,E1 242.948} C_DIS
LIN {X 0.041,Y -162.200,Z 1011.321,A 0.000,B 0.000,C 90.000,E1 237.709} C_DIS
LIN {X 0.009,Y -160.773,Z 1011.311,A 0.000,B 0.000,C 90.000,E1 235.960} C_DIS
LIN {X -0.019,Y -157.568,Z 1011.291,A 0.000,B 0.000,C 90.000,E1 232.431} C_DIS
LIN {X 0.014,Y -155.598,Z 1011.276,A 0.000,B 0.000,C 90.000,E1 229.747} C_DIS
LIN {X 0.065,Y -151.879,Z 1011.251,A 0.000,B 0.000,C 90.000,E1 225.243} C_DIS
LIN {X 0.078,Y -150.106,Z 1011.236,A 0.000,B 0.000,C 90.000,E1 222.528} C_DIS
LIN {X -0.004,Y -146.902,Z 1011.211,A 0.000,B 0.000,C 90.000,E1 218.016} C_DIS
LIN {X 0.016,Y -145.489,Z 1011.196,A 0.000,B 0.000,C 90.000,E1 215.264} C_DIS
LIN {X 0.016,Y -142.896,Z 1011.170,A 0.000,B 0.000,C 90.000,E1 210.669} C_DIS
LIN {X -0.054,Y -141.517,Z 1011.150,A 0.000,B 0.000,C 90.000,E1 207.001} C_DIS
LIN {X -0.010,Y -139.394,Z 1011.114,A 0.000,B 0.000,C 90.000,E1 200.482} C_DIS
LIN {X 0.040,Y -139.104,Z 1011.103,A 0.000,B 0.000,C 90.000,E1 198.598} C_DIS
LIN {X 0.033,Y -138.353,Z 1011.057,A 0.000,B 0.000,C 90.000,E1 190.197} C_DIS
LIN {X 0.026,Y -139.512,Z 1011.005,A 0.000,B 0.000,C 90.000,E1 180.859} C_DIS
LIN {X -0.034,Y -141.159,Z 1010.974,A 0.000,B 0.000,C 90.000,E1 175.298} C_DIS
LIN {X 0.078,Y -142.539,Z 1010.958,A 0.000,B 0.000,C 90.000,E1 172.470} C_DIS
LIN {X 0.004,Y -144.809,Z 1010.933,A 0.000,B 0.000,C 90.000,E1 167.881} C_DIS
LIN {X -0.008,Y -147.429,Z 1010.912,A 0.000,B 0.000,C 90.000,E1 164.212} C_DIS
LIN {X 0.021,Y -150.008,Z 1010.892,A 0.000,B 0.000,C 90.000,E1 160.550} C_DIS
LIN {X 0.028,Y -153.340,Z 1010.872,A 0.000,B 0.000,C 90.000,E1 156.922} C_DIS
LIN {X 0.010,Y -155.874,Z 1010.857,A 0.000,B 0.000,C 90.000,E1 154.229} C_DIS
LIN {X -0.024,Y -159.729,Z 1010.837,A 0.000,B 0.000,C 90.000,E1 150.667} C_DIS
LIN {X 0.043,Y -161.968,Z 1010.827,A 0.000,B 0.000,C 90.000,E1 148.869} C_DIS
LIN {X -0.074,Y -166.160,Z 1010.808,A 0.000,B 0.000,C 90.000,E1 145.388} C_DIS
LIN {X -0.078,Y -171.173,Z 1010.788,A 0.000,B 0.000,C 90.000,E1 141.904} C_DIS
LIN {X -0.044,Y -176.054,Z 1010.769,A 0.000,B 0.000,C 90.000,E1 138.447} C_DIS
LIN {X -0.049,Y -180.310,Z 1010.755,A 0.000,B 0.000,C 90.000,E1 135.891} C_DIS
LIN {X -0.078,Y -185.721,Z 1010.736,A 0.000,B 0.000,C 90.000,E1 132.528} C_DIS
LIN {X -0.027,Y -190.328,Z 1010.722,A 0.000,B 0.000,C 90.000,E1 130.011} C_DIS
LIN {X -0.077,Y -196.515,Z 1010.703,A 0.000,B 0.000,C 90.000,E1 126.503} C_DIS
LIN {X 0.076,Y -301.599,Z 1010.703,A 0.000,B 0.000,C 90.000,E1 126.457} C_DIS
LIN {X -0.070,Y -303.051,Z 1010.702,A 0.000,B 0.000,C 90.000,E1 126.457} C_DIS
LIN {X -0.019,Y -308.355,Z 1010.701,A 0.000,B 0.000,C 90.000,E1 126.171} C_DIS
LIN {X 0.034,Y -311.180,Z 1010.699,A 0.000,B 0.000,C 90.000,E1 125.884} C_DIS
LIN {X 0.138,Y -314.867,Z 1010.696,A 0.000,B 0.000,C 90.000,E1 125.311} C_DIS
LIN {X -0.071,Y -316.375,Z 1010.695,A 0.000,B 0.000,C 90.000,E1 125.025} C_DIS
LIN {X 0.030,Y -319.625,Z 1010.689,A 0.000,B 0.000,C 90.000,E1 124.040} C_DIS
LIN {X -0.044,Y -330.874,Z 1010.672,A 0.000,B 0.000,C 90.000,E1 120.875} C_DIS
LIN {X 0.060,Y -342.399,Z 1010.656,A 0.000,B 0.000,C 90.000,E1 118.052} C_DIS
LIN {X -0.145,Y -355.359,Z 1010.641,A 0.000,B 0.000,C 90.000,E1 115.335} C_DIS
LIN {X 0.130,Y -368.173,Z 1010.627,A 0.000,B 0.000,C 90.000,E1 112.898} C_DIS
LIN {X 0.119,Y -382.300,Z 1010.614,A 0.000,B 0.000,C 90.000,E1 110.556} C_DIS
LIN {X -0.050,Y -397.840,Z 1010.602,A 0.000,B 0.000,C 90.000,E1 108.290} C_DIS
LIN {X 0.169,Y -414.903,Z 1010.589,A 0.000,B 0.000,C 90.000,E1 106.024} C_DIS
LIN {X -0.101,Y -433.613,Z 1010.577,A 0.000,B 0.000,C 90.000,E1 103.883} C_DIS
LIN {X -0.176,Y -453.575,Z 1010.566,A 0.000,B 0.000,C 90.000,E1 101.827} C_DIS
LIN {X 0.000,Y -466.327,Z 1010.559,A 0.000,B 0.000,C 90.000,E1 100.602} C_DIS
LIN {X 0.012,Y -468.631,Z 1010.558,A 0.000,B 0.000,C 90.000,E1 100.366} C_DIS
LIN {X -0.192,Y -470.469,Z 1010.556,A 0.000,B 0.000,C 90.000,E1 100.141} C_DIS
LIN {X 0.152,Y -471.854,Z 1010.555,A 0.000,B 0.000,C 90.000,E1 99.849} C_DIS
LIN {X -0.137,Y -473.638,Z 1010.552,A 0.000,B 0.000,C 90.000,E1 99.378} C_DIS
LIN {X -0.029,Y -474.338,Z 1010.549,A 0.000,B 0.000,C 90.000,E1 98.859} C_DIS
LIN {X 0.093,Y -474.069,Z 1010.546,A 0.000,B 0.000,C 90.000,E1 98.341} C_DIS
LIN {X -0.182,Y -472.797,Z 1010.544,A 0.000,B 0.000,C 90.000,E1 97.871} C_DIS
LIN {X 0.082,Y -471.725,Z 1010.542,A 0.000,B 0.000,C 90.000,E1 97.587} C_DIS
LIN {X -0.059,Y -470.288,Z 1010.541,A 0.000,B 0.000,C 90.000,E1 97.352} C_DIS
LIN {X -0.010,Y -458.053,Z 1010.531,A 0.000,B 0.000,C 90.000,E1 95.568} C_DIS
LIN {X -0.006,Y -443.885,Z 1010.519,A 0.000,B 0.000,C 90.000,E1 93.498} C_DIS
LIN {X -0.062,Y -427.281,Z 1010.505,A 0.000,B 0.000,C 90.000,E1 90.859} C_DIS
LIN {X -0.074,Y -410.813,Z 1010.488,A 0.000,B 0.000,C 90.000,E1 87.879} C_DIS
LIN {X -0.041,Y -401.986,Z 1010.479,A 0.000,B 0.000,C 90.000,E1 86.216} C_DIS
LIN {X -0.092,Y -391.349,Z 1010.468,A 0.000,B 0.000,C 90.000,E1 84.261} C_DIS
LIN {X 0.035,Y -382.063,Z 1010.459,A 0.000,B 0.000,C 90.000,E1 82.534} C_DIS
LIN {X 0.089,Y -372.461,Z 1010.449,A 0.000,B 0.000,C 90.000,E1 80.792} C_DIS
LIN {X -0.049,Y -360.886,Z 1010.438,A 0.000,B 0.000,C 90.000,E1 78.757} C_DIS
LIN {X -0.005,Y -347.636,Z 1010.424,A 0.000,B 0.000,C 90.000,E1 76.353} C_DIS
LIN {X -0.134,Y -333.182,Z 1010.409,A 0.000,B 0.000,C 90.000,E1 73.614} C_DIS
LIN {X -0.078,Y -320.780,Z 1010.395,A 0.000,B 0.000,C 90.000,E1 71.094} C_DIS
LIN {X -0.128,Y -308.618,Z 1010.381,A 0.000,B 0.000,C 90.000,E1 68.539} C_DIS
LIN {X 0.138,Y -295.298,Z 1010.364,A 0.000,B 0.000,C 90.000,E1 65.537} C_DIS
LIN {X 0.043,Y -283.809,Z 1010.349,A 0.000,B 0.000,C 90.000,E1 62.871} C_DIS
LIN {X 0.109,Y -273.885,Z 1010.336,A 0.000,B 0.000,C 90.000,E1 60.461} C_DIS
LIN {X 0.004,Y -264.107,Z 1010.322,A 0.000,B 0.000,C 90.000,E1 58.043} C_DIS
LIN {X -0.045,Y -251.933,Z 1010.305,A 0.000,B 0.000,C 90.000,E1 54.848} C_DIS
LIN {X 0.083,Y -240.392,Z 1010.286,A 0.000,B 0.000,C 90.000,E1 51.537} C_DIS
LIN {X 0.148,Y -229.544,Z 1010.268,A 0.000,B 0.000,C 90.000,E1 48.162} C_DIS
LIN {X 0.040,Y -219.311,Z 1010.249,A 0.000,B 0.000,C 90.000,E1 44.757} C_DIS
LIN {X -0.068,Y -210.654,Z 1010.231,A 0.000,B 0.000,C 90.000,E1 41.676} C_DIS
LIN {X 0.113,Y -202.542,Z 1010.214,A 0.000,B 0.000,C 90.000,E1 38.463} C_DIS
LIN {X -0.119,Y -195.040,Z 1010.196,A 0.000,B 0.000,C 90.000,E1 35.311} C_DIS
LIN {X -0.003,Y -188.360,Z 1010.178,A 0.000,B 0.000,C 90.000,E1 32.005} C_DIS
LIN {X -0.029,Y -182.496,Z 1010.159,A 0.000,B 0.000,C 90.000,E1 28.693} C_DIS
LIN {X -0.050,Y -177.438,Z 1010.141,A 0.000,B 0.000,C 90.000,E1 25.335} C_DIS
LIN {X 0.056,Y -173.105,Z 1010.122,A 0.000,B 0.000,C 90.000,E1 21.897} C_DIS
LIN {X -0.031,Y -169.513,Z 1010.103,A 0.000,B 0.000,C 90.000,E1 18.489} C_DIS
LIN {X 0.067,Y -165.955,Z 1010.079,A 0.000,B 0.000,C 90.000,E1 14.120} C_DIS
LIN {X -0.059,Y -163.133,Z 1010.049,A 0.000,B 0.000,C 90.000,E1 8.916} C_DIS
LIN {X 0.006,Y -163.906,Z 1009.953,A 0.000,B 0.000,C 90.000,E1 351.602} C_DIS
LIN {X -0.016,Y -166.462,Z 1009.929,A 0.000,B 0.000,C 90.000,E1 347.229} C_DIS
LIN {X 0.059,Y -170.084,Z 1009.905,A 0.000,B 0.000,C 90.000,E1 342.851} C_DIS
LIN {X 0.080,Y -173.836,Z 1009.886,A 0.000,B 0.000,C 90.000,E1 339.390} C_DIS
LIN {X -0.010,Y -178.474,Z 1009.867,A 0.000,B 0.000,C 90.000,E1 335.997} C_DIS
LIN {X -0.022,Y -183.866,Z 1009.848,A 0.000,B 0.000,C 90.000,E1 332.615} C_DIS
LIN {X -0.056,Y -190.070,Z 1009.829,A 0.000,B 0.000,C 90.000,E1 329.282} C_DIS
LIN {X 0.029,Y -196.926,Z 1009.811,A 0.000,B 0.000,C 90.000,E1 325.960} C_DIS
LIN {X 0.020,Y -204.331,Z 1009.793,A 0.000,B 0.000,C 90.000,E1 322.718} C_DIS
LIN {X 0.011,Y -213.438,Z 1009.773,A 0.000,B 0.000,C 90.000,E1 319.138} C_DIS
LIN {X -0.140,Y -221.977,Z 1009.756,A 0.000,B 0.000,C 90.000,E1 316.053} C_DIS
LIN {X 0.074,Y -231.336,Z 1009.739,A 0.000,B 0.000,C 90.000,E1 312.933} C_DIS
LIN {X 0.029,Y -236.615,Z 1009.730,A 0.000,B 0.000,C 90.000,E1 311.434} C_DIS
LIN {X 0.048,Y -244.042,Z 1009.720,A 0.000,B 0.000,C 90.000,E1 309.564} C_DIS
LIN {X 0.039,Y -252.388,Z 1009.710,A 0.000,B 0.000,C 90.000,E1 307.729} C_DIS
LIN {X -0.107,Y -263.567,Z 1009.698,A 0.000,B 0.000,C 90.000,E1 305.598} C_DIS
LIN {X 0.051,Y -280.001,Z 1009.682,A 0.000,B 0.000,C 90.000,E1 302.752} C_DIS
LIN {X -0.053,Y -295.407,Z 1009.669,A 0.000,B 0.000,C 90.000,E1 300.384} C_DIS
LIN {X 0.046,Y -314.312,Z 1009.654,A 0.000,B 0.000,C 90.000,E1 297.719} C_DIS
LIN {X 0.066,Y -329.912,Z 1009.643,A 0.000,B 0.000,C 90.000,E1 295.796} C_DIS
LIN {X -0.138,Y -351.570,Z 1009.630,A 0.000,B 0.000,C 90.000,E1 293.515} C_DIS
LIN {X -0.117,Y -373.465,Z 1009.619,A 0.000,B 0.000,C 90.000,E1 291.408} C_DIS
LIN {X 0.151,Y -389.666,Z 1009.611,A 0.000,B 0.000,C 90.000,E1 289.885} C_DIS
LIN {X 0.084,Y -400.527,Z 1009.605,A 0.000,B 0.000,C 90.000,E1 288.906} C_DIS
LIN {X -0.156,Y -411.114,Z 1009.600,A 0.000,B 0.000,C 90.000,E1 287.946} C_DIS
LIN {X -0.023,Y -418.763,Z 1009.595,A 0.000,B 0.000,C 90.000,E1 287.166} C_DIS
LIN {X -0.012,Y -428.547,Z 1009.590,A 0.000,B 0.000,C 90.000,E1 286.134} C_DIS
LIN {X -0.017,Y -438.124,Z 1009.584,A 0.000,B 0.000,C 90.000,E1 285.064} C_DIS
LIN {X -0.256,Y -449.221,Z 1009.576,A 0.000,B 0.000,C 90.000,E1 283.772} C_DIS
LIN {X -0.047,Y -457.382,Z 1009.571,A 0.000,B 0.000,C 90.000,E1 282.703} C_DIS
LIN {X -0.222,Y -462.996,Z 1009.566,A 0.000,B 0.000,C 90.000,E1 281.951} C_DIS
LIN {X 0.052,Y -469.684,Z 1009.561,A 0.000,B 0.000,C 90.000,E1 280.894} C_DIS
LIN {X -0.011,Y -474.142,Z 1009.556,A 0.000,B 0.000,C 90.000,E1 280.141} C_DIS
LIN {X 0.052,Y -477.992,Z 1009.552,A 0.000,B 0.000,C 90.000,E1 279.378} C_DIS
LIN {X 0.062,Y -481.184,Z 1009.548,A 0.000,B 0.000,C 90.000,E1 278.624} C_DIS
LIN {X 0.223,Y -482.980,Z 1009.545,A 0.000,B 0.000,C 90.000,E1 278.106} C_DIS
LIN {X -0.085,Y -484.528,Z 1009.542,A 0.000,B 0.000,C 90.000,E1 277.644} C_DIS
LIN {X 0.096,Y -485.825,Z 1009.540,A 0.000,B 0.000,C 90.000,E1 277.125} C_DIS
LIN {X -0.196,Y -486.918,Z 1009.537,A 0.000,B 0.000,C 90.000,E1 276.663} C_DIS
LIN {X 0.003,Y -487.779,Z 1009.534,A 0.000,B 0.000,C 90.000,E1 276.144} C_DIS
LIN {X 0.209,Y -488.399,Z 1009.531,A 0.000,B 0.000,C 90.000,E1 275.625} C_DIS
LIN {X -0.068,Y -488.656,Z 1009.529,A 0.000,B 0.000,C 90.000,E1 275.163} C_DIS
LIN {X 0.143,Y -488.486,Z 1009.526,A 0.000,B 0.000,C 90.000,E1 274.645} C_DIS
LIN {X -0.168,Y -487.811,Z 1009.523,A 0.000,B 0.000,C 90.000,E1 274.188} C_DIS
LIN {X 0.042,Y -486.661,Z 1009.520,A 0.000,B 0.000,C 90.000,E1 273.669} C_DIS
LIN {X 0.217,Y -484.919,Z 1009.518,A 0.000,B 0.000,C 90.000,E1 273.154} C_DIS
LIN {X -0.072,Y -482.479,Z 1009.515,A 0.000,B 0.000,C 90.000,E1 272.694} C_DIS
LIN {X 0.082,Y -479.297,Z 1009.512,A 0.000,B 0.000,C 90.000,E1 272.178} C_DIS
LIN {X 0.235,Y -475.289,Z 1009.509,A 0.000,B 0.000,C 90.000,E1 271.661} C_DIS
LIN {X -0.122,Y -470.343,Z 1009.507,A 0.000,B 0.000,C 90.000,E1 271.203} C_DIS
LIN {X 0.156,Y -464.560,Z 1009.504,A 0.000,B 0.000,C 90.000,E1 270.688} C_DIS
LIN {X -0.060,Y -458.352,Z 1009.502,A 0.000,B 0.000,C 90.000,E1 270.286} C_DIS
LIN {X -0.170,Y -455.240,Z 1009.500,A 0.000,B 0.000,C 90.000,E1 270.115} C_DIS
LIN {X -0.122,Y -448.319,Z 1009.499,A 0.000,B 0.000,C 90.000,E1 269.771} C_DIS
LIN {X -0.029,Y -441.133,Z 1009.497,A 0.000,B 0.000,C 90.000,E1 269.484} C_DIS
LIN {X 0.051,Y -433.576,Z 1009.496,A 0.000,B 0.000,C 90.000,E1 269.255} C_DIS
LIN {X 0.093,Y -425.337,Z 1009.495,A 0.000,B 0.000,C 90.000,E1 269.083} C_DIS
LIN {X 0.052,Y -416.558,Z 1009.494,A 0.000,B 0.000,C 90.000,E1 268.969} C_DIS
LIN {X 0.097,Y -402.345,Z 1009.494,A 0.000,B 0.000,C 90.000,E1 268.854} C_DIS
LIN {X 0.030,Y -400.382,Z 1009.494,A 0.000,B 0.000,C 90.000,E1 268.854} C_DIS
LIN {X -0.017,Y -181.286,Z 1009.494,A 0.000,B 0.000,C 90.000,E1 268.854} C_DIS
LIN {X 0.046,Y -180.887,Z 1009.473,A 0.000,B 0.000,C 90.000,E1 265.122} C_DIS
LIN {X -0.071,Y -179.010,Z 1009.445,A 0.000,B 0.000,C 90.000,E1 260.095} C_DIS
LIN {X 0.023,Y -178.625,Z 1009.440,A 0.000,B 0.000,C 90.000,E1 259.218} C_DIS
LIN {X -0.079,Y -175.677,Z 1009.412,A 0.000,B 0.000,C 90.000,E1 254.157} C_DIS
LIN {X -0.066,Y -172.393,Z 1009.388,A 0.000,B 0.000,C 90.000,E1 249.880} C_DIS
LIN {X -0.050,Y -171.199,Z 1009.379,A 0.000,B 0.000,C 90.000,E1 248.156} C_DIS
LIN {X 0.001,Y -167.488,Z 1009.355,A 0.000,B 0.000,C 90.000,E1 243.819} C_DIS
LIN {X 0.009,Y -166.884,Z 1009.350,A 0.000,B 0.000,C 90.000,E1 242.948} C_DIS
LIN {X 0.000,Y -162.189,Z 1009.321,A 0.000,B 0.000,C 90.000,E1 237.709} C_DIS
LIN {X -0.032,Y -160.759,Z 1009.311,A 0.000,B 0.000,C 90.000,E1 235.960} C_DIS
LIN {X 0.036,Y -157.556,Z 1009.291,A 0.000,B 0.000,C 90.000,E1 232.396} C_DIS
LIN {X -0.026,Y -155.584,Z 1009.276,A 0.000,B 0.000,C 90.000,E1 229.747} C_DIS
LIN {X 0.025,Y -151.869,Z 1009.251,A 0.000,B 0.000,C 90.000,E1 225.243} C_DIS
LIN {X 0.039,Y -150.093,Z 1009.236,A 0.000,B 0.000,C 90.000,E1 222.528} C_DIS
LIN {X -0.043,Y -146.893,Z 1009.211,A 0.000,B 0.000,C 90.000,E1 218.016} C_DIS
LIN {X 0.061,Y -145.480,Z 1009.196,A 0.000,B 0.000,C 90.000,E1 215.231} C_DIS
LIN {X -0.023,Y -142.889,Z 1009.170,A 0.000,B 0.000,C 90.000,E1 210.669} C_DIS
LIN {X 0.034,Y -141.509,Z 1009.150,A 0.000,B 0.000,C 90.000,E1 206.950} C_DIS
LIN {X -0.048,Y -139.392,Z 1009.114,A 0.000,B 0.000,C 90.000,E1 200.482} C_DIS
LIN {X 0.003,Y -139.099,Z 1009.103,A 0.000,B 0.000,C 90.000,E1 198.598} C_DIS
LIN {X -0.005,Y -138.354,Z 1009.057,A 0.000,B 0.000,C 90.000,E1 190.197} C_DIS
LIN {X -0.012,Y -139.515,Z 1009.005,A 0.000,B 0.000,C 90.000,E1 180.859} C_DIS
LIN {X -0.072,Y -141.165,Z 1008.974,A 0.000,B 0.000,C 90.000,E1 175.298} C_DIS
LIN {X 0.040,Y -142.545,Z 1008.958,A 0.000,B 0.000,C 90.000,E1 172.470} C_DIS
LIN {X -0.034,Y -144.818,Z 1008.933,A 0.000,B 0.000,C 90.000,E1 167.881} C_DIS
LIN {X -0.047,Y -147.440,Z 1008.912,A 0.000,B 0.000,C 90.000,E1 164.212} C_DIS
LIN {X -0.019,Y -150.020,Z 1008.892,A 0.000,B 0.000,C 90.000,E1 160.550} C_DIS
LIN {X -0.012,Y -153.355,Z 1008.872,A 0.000,B 0.000,C 90.000,E1 156.922} C_DIS
LIN {X 0.036,Y -155.889,Z 1008.857,A 0.000,B 0.000,C 90.000,E1 154.204} C_DIS
LIN {X -0.065,Y -159.747,Z 1008.837,A 0.000,B 0.000,C 90.000,E1 150.667} C_DIS
LIN {X 0.001,Y -161.986,Z 1008.827,A 0.000,B 0.000,C 90.000,E1 148.869} C_DIS
LIN {X 0.021,Y -166.178,Z 1008.807,A 0.000,B 0.000,C 90.000,E1 145.341} C_DIS
LIN {X 0.014,Y -171.193,Z 1008.788,A 0.000,B 0.000,C 90.000,E1 141.859} C_DIS
LIN {X 0.044,Y -176.075,Z 1008.769,A 0.000,B 0.000,C 90.000,E1 138.405} C_DIS
LIN {X -0.094,Y -180.335,Z 1008.755,A 0.000,B 0.000,C 90.000,E1 135.891} C_DIS
LIN {X 0.014,Y -185.745,Z 1008.736,A 0.000,B 0.000,C 90.000,E1 132.486} C_DIS
LIN {X -0.072,Y -190.356,Z 1008.722,A 0.000,B 0.000,C 90.000,E1 130.011} C_DIS
LIN {X 0.069,Y -196.435,Z 1008.703,A 0.000,B 0.000,C 90.000,E1 126.503} C_DIS
LIN {X 0.054,Y -301.037,Z 1008.703,A 0.000,B 0.000,C 90.000,E1 126.503} C_DIS
LIN {X -0.046,Y -302.350,Z 1008.703,A 0.000,B 0.000,C 90.000,E1 126.503} C_DIS
LIN {X -0.016,Y -306.260,Z 1008.702,A 0.000,B 0.000,C 90.000,E1 126.343} C_DIS
LIN {X 0.080,Y -308.445,Z 1008.701,A 0.000,B 0.000,C 90.000,E1 126.171} C_DIS
LIN {X -0.040,Y -311.464,Z 1008.699,A 0.000,B 0.000,C 90.000,E1 125.884} C_DIS
LIN {X -0.041,Y -315.084,Z 1008.696,A 0.000,B 0.000,C 90.000,E1 125.311} C_DIS
LIN {X 0.010,Y -316.516,Z 1008.694,A 0.000,B 0.000,C 90.000,E1 124.978} C_DIS
LIN {X 0.118,Y -329.774,Z 1008.673,A 0.000,B 0.000,C 90.000,E1 121.131} C_DIS
LIN {X -0.113,Y -341.164,Z 1008.657,A 0.000,B 0.000,C 90.000,E1 118.359} C_DIS
LIN {X -0.044,Y -353.972,Z 1008.642,A 0.000,B 0.000,C 90.000,E1 115.591} C_DIS
LIN {X -0.137,Y -366.644,Z 1008.629,A 0.000,B 0.000,C 90.000,E1 113.206} C_DIS
LIN {X -0.062,Y -380.618,Z 1008.616,A 0.000,B 0.000,C 90.000,E1 110.844} C_DIS
LIN {X -0.041,Y -395.992,Z 1008.603,A 0.000,B 0.000,C 90.000,E1 108.544} C_DIS
LIN {X -0.139,Y -412.878,Z 1008.591,A 0.000,B 0.000,C 90.000,E1 106.315} C_DIS
LIN {X -0.058,Y -431.396,Z 1008.578,A 0.000,B 0.000,C 90.000,E1 104.120} C_DIS
LIN {X 0.173,Y -451.264,Z 1008.567,A 0.000,B 0.000,C 90.000,E1 102.007} C_DIS
LIN {X -0.195,Y -466.562,Z 1008.559,A 0.000,B 0.000,C 90.000,E1 100.602} C_DIS
LIN {X -0.184,Y -468.807,Z 1008.557,A 0.000,B 0.000,C 90.000,E1 100.366} C_DIS
LIN {X 0.128,Y -470.623,Z 1008.556,A 0.000,B 0.000,C 90.000,E1 100.074} C_DIS
LIN {X -0.105,Y -471.986,Z 1008.555,A 0.000,B 0.000,C 90.000,E1 99.849} C_DIS
LIN {X 0.074,Y -473.703,Z 1008.552,A 0.000,B 0.000,C 90.000,E1 99.321} C_DIS
LIN {X 0.184,Y -474.346,Z 1008.549,A 0.000,B 0.000,C 90.000,E1 98.803} C_DIS
LIN {X -0.162,Y -474.022,Z 1008.546,A 0.000,B 0.000,C 90.000,E1 98.341} C_DIS
LIN {X 0.031,Y -472.690,Z 1008.543,A 0.000,B 0.000,C 90.000,E1 97.814} C_DIS
LIN {X -0.172,Y -471.579,Z 1008.542,A 0.000,B 0.000,C 90.000,E1 97.587} C_DIS
LIN {X 0.154,Y -470.095,Z 1008.541,A 0.000,B 0.000,C 90.000,E1 97.296} C_DIS
LIN {X 0.196,Y -457.881,Z 1008.531,A 0.000,B 0.000,C 90.000,E1 95.511} C_DIS
LIN {X 0.143,Y -440.295,Z 1008.516,A 0.000,B 0.000,C 90.000,E1 92.922} C_DIS
LIN {X -0.164,Y -425.566,Z 1008.503,A 0.000,B 0.000,C 90.000,E1 90.573} C_DIS
LIN {X 0.099,Y -410.662,Z 1008.488,A 0.000,B 0.000,C 90.000,E1 87.822} C_DIS
LIN {X 0.125,Y -401.829,Z 1008.479,A 0.000,B 0.000,C 90.000,E1 86.159} C_DIS
LIN {X 0.050,Y -392.722,Z 1008.469,A 0.000,B 0.000,C 90.000,E1 84.489} C_DIS
LIN {X -0.177,Y -383.478,Z 1008.460,A 0.000,B 0.000,C 90.000,E1 82.818} C_DIS
LIN {X -0.143,Y -373.916,Z 1008.450,A 0.000,B 0.000,C 90.000,E1 81.084} C_DIS
LIN {X 0.131,Y -364.020,Z 1008.441,A 0.000,B 0.000,C 90.000,E1 79.285} C_DIS
LIN {X -0.048,Y -352.366,Z 1008.429,A 0.000,B 0.000,C 90.000,E1 77.229} C_DIS
LIN {X -0.123,Y -339.335,Z 1008.416,A 0.000,B 0.000,C 90.000,E1 74.810} C_DIS
LIN {X -0.053,Y -325.243,Z 1008.400,A 0.000,B 0.000,C 90.000,E1 72.000} C_DIS
LIN {X 0.008,Y -312.978,Z 1008.386,A 0.000,B 0.000,C 90.000,E1 69.444} C_DIS
LIN {X -0.023,Y -302.452,Z 1008.373,A 0.000,B 0.000,C 90.000,E1 67.177} C_DIS
LIN {X 0.071,Y -292.241,Z 1008.360,A 0.000,B 0.000,C 90.000,E1 64.845} C_DIS
LIN {X 0.063,Y -282.236,Z 1008.347,A 0.000,B 0.000,C 90.000,E1 62.487} C_DIS
LIN {X 0.097,Y -272.324,Z 1008.334,A 0.000,B 0.000,C 90.000,E1 60.078} C_DIS
LIN {X 0.004,Y -261.153,Z 1008.318,A 0.000,B 0.000,C 90.000,E1 57.296} C_DIS
LIN {X 0.014,Y -249.151,Z 1008.300,A 0.000,B 0.000,C 90.000,E1 54.069} C_DIS
LIN {X -0.125,Y -237.756,Z 1008.282,A 0.000,B 0.000,C 90.000,E1 50.803} C_DIS
LIN {X 0.025,Y -227.042,Z 1008.263,A 0.000,B 0.000,C 90.000,E1 47.391} C_DIS
LIN {X 0.005,Y -216.885,Z 1008.244,A 0.000,B 0.000,C 90.000,E1 43.947} C_DIS
LIN {X -0.002,Y -208.394,Z 1008.227,A 0.000,B 0.000,C 90.000,E1 40.825} C_DIS
LIN {X -0.009,Y -200.420,Z 1008.209,A 0.000,B 0.000,C 90.000,E1 37.649} C_DIS
LIN {X 0.025,Y -193.148,Z 1008.191,A 0.000,B 0.000,C 90.000,E1 34.405} C_DIS
LIN {X -0.012,Y -186.684,Z 1008.173,A 0.000,B 0.000,C 90.000,E1 31.131} C_DIS
LIN {X 0.078,Y -181.060,Z 1008.154,A 0.000,B 0.000,C 90.000,E1 27.769} C_DIS
LIN {X 0.097,Y -176.198,Z 1008.136,A 0.000,B 0.000,C 90.000,E1 24.387} C_DIS
LIN {X 0.102,Y -172.068,Z 1008.117,A 0.000,B 0.000,C 90.000,E1 20.972} C_DIS
LIN {X -0.067,Y -168.647,Z 1008.098,A 0.000,B 0.000,C 90.000,E1 17.583} C_DIS
LIN {X -0.042,Y -165.342,Z 1008.073,A 0.000,B 0.000,C 90.000,E1 13.231} C_DIS
LIN {X -0.088,Y -162.791,Z 1008.044,A 0.000,B 0.000,C 90.000,E1 7.992} C_DIS
LIN {X 0.038,Y -163.487,Z 1007.958,A 0.000,B 0.000,C 90.000,E1 352.470} C_DIS
LIN {X -0.017,Y -166.451,Z 1007.929,A 0.000,B 0.000,C 90.000,E1 347.229} C_DIS
LIN {X 0.058,Y -170.083,Z 1007.905,A 0.000,B 0.000,C 90.000,E1 342.851} C_DIS
LIN {X 0.079,Y -173.840,Z 1007.886,A 0.000,B 0.000,C 90.000,E1 339.390} C_DIS
LIN {X 0.062,Y -178.496,Z 1007.867,A 0.000,B 0.000,C 90.000,E1 335.973} C_DIS
LIN {X -0.023,Y -183.897,Z 1007.848,A 0.000,B 0.000,C 90.000,E1 332.615} C_DIS
LIN {X -0.056,Y -190.107,Z 1007.829,A 0.000,B 0.000,C 90.000,E1 329.282} C_DIS
LIN {X 0.030,Y -196.958,Z 1007.811,A 0.000,B 0.000,C 90.000,E1 325.960} C_DIS
LIN {X 0.022,Y -204.369,Z 1007.793,A 0.000,B 0.000,C 90.000,E1 322.718} C_DIS
LIN {X 0.014,Y -213.452,Z 1007.773,A 0.000,B 0.000,C 90.000,E1 319.138} C_DIS
LIN {X -0.137,Y -221.980,Z 1007.756,A 0.000,B 0.000,C 90.000,E1 316.053} C_DIS
LIN {X 0.078,Y -231.291,Z 1007.739,A 0.000,B 0.000,C 90.000,E1 312.933} C_DIS
LIN {X 0.031,Y -236.570,Z 1007.730,A 0.000,B 0.000,C 90.000,E1 311.434} C_DIS
LIN {X 0.051,Y -244.056,Z 1007.720,A 0.000,B 0.000,C 90.000,E1 309.564} C_DIS
LIN {X 0.043,Y -252.436,Z 1007.710,A 0.000,B 0.000,C 90.000,E1 307.729} C_DIS
LIN {X -0.103,Y -263.627,Z 1007.698,A 0.000,B 0.000,C 90.000,E1 305.598} C_DIS
LIN {X 0.056,Y -280.051,Z 1007.682,A 0.000,B 0.000,C 90.000,E1 302.752} C_DIS
LIN {X -0.045,Y -295.475,Z 1007.669,A 0.000,B 0.000,C 90.000,E1 300.384} C_DIS
LIN {X 0.057,Y -314.386,Z 1007.654,A 0.000,B 0.000,C 90.000,E1 297.719} C_DIS
LIN {X 0.093,Y -330.004,Z 1007.643,A 0.000,B 0.000,C 90.000,E1 295.796} C_DIS
LIN {X 0.037,Y -351.932,Z 1007.630,A 0.000,B 0.000,C 90.000,E1 293.462} C_DIS
LIN {X 0.103,Y -373.794,Z 1007.619,A 0.000,B 0.000,C 90.000,E1 291.354} C_DIS
LIN {X -0.060,Y -390.275,Z 1007.610,A 0.000,B 0.000,C 90.000,E1 289.866} C_DIS
LIN {X 0.102,Y -401.107,Z 1007.605,A 0.000,B 0.000,C 90.000,E1 288.852} C_DIS
LIN {X -0.047,Y -411.680,Z 1007.599,A 0.000,B 0.000,C 90.000,E1 287.873} C_DIS
LIN {X -0.088,Y -421.774,Z 1007.594,A 0.000,B 0.000,C 90.000,E1 286.858} C_DIS
LIN {X 0.008,Y -431.610,Z 1007.588,A 0.000,B 0.000,C 90.000,E1 285.788} C_DIS
LIN {X 0.016,Y -440.930,Z 1007.582,A 0.000,B 0.000,C 90.000,E1 284.717} C_DIS
LIN {X 0.134,Y -449.708,Z 1007.576,A 0.000,B 0.000,C 90.000,E1 283.647} C_DIS
LIN {X -0.195,Y -457.835,Z 1007.570,A 0.000,B 0.000,C 90.000,E1 282.647} C_DIS
LIN {X 0.182,Y -463.408,Z 1007.566,A 0.000,B 0.000,C 90.000,E1 281.827} C_DIS
LIN {X -0.088,Y -470.070,Z 1007.560,A 0.000,B 0.000,C 90.000,E1 280.838} C_DIS
LIN {X -0.065,Y -474.508,Z 1007.556,A 0.000,B 0.000,C 90.000,E1 280.074} C_DIS
LIN {X -0.082,Y -478.341,Z 1007.552,A 0.000,B 0.000,C 90.000,E1 279.321} C_DIS
LIN {X -0.068,Y -481.508,Z 1007.548,A 0.000,B 0.000,C 90.000,E1 278.568} C_DIS
LIN {X 0.095,Y -483.269,Z 1007.545,A 0.000,B 0.000,C 90.000,E1 278.049} C_DIS
LIN {X -0.213,Y -484.797,Z 1007.542,A 0.000,B 0.000,C 90.000,E1 277.587} C_DIS
LIN {X -0.029,Y -486.102,Z 1007.539,A 0.000,B 0.000,C 90.000,E1 277.068} C_DIS
LIN {X 0.165,Y -487.150,Z 1007.536,A 0.000,B 0.000,C 90.000,E1 276.549} C_DIS
LIN {X -0.118,Y -488.002,Z 1007.534,A 0.000,B 0.000,C 90.000,E1 276.087} C_DIS
LIN {X 0.090,Y -488.548,Z 1007.531,A 0.000,B 0.000,C 90.000,E1 275.568} C_DIS
LIN {X -0.185,Y -488.744,Z 1007.528,A 0.000,B 0.000,C 90.000,E1 275.106} C_DIS
LIN {X 0.027,Y -488.535,Z 1007.526,A 0.000,B 0.000,C 90.000,E1 274.588} C_DIS
LIN {X 0.203,Y -487.837,Z 1007.523,A 0.000,B 0.000,C 90.000,E1 274.073} C_DIS
LIN {X -0.072,Y -486.617,Z 1007.520,A 0.000,B 0.000,C 90.000,E1 273.612} C_DIS
LIN {X 0.129,Y -484.799,Z 1007.517,A 0.000,B 0.000,C 90.000,E1 273.094} C_DIS
LIN {X -0.185,Y -482.272,Z 1007.515,A 0.000,B 0.000,C 90.000,E1 272.636} C_DIS
LIN {X -0.031,Y -479.008,Z 1007.512,A 0.000,B 0.000,C 90.000,E1 272.121} C_DIS
LIN {X -0.200,Y -477.095,Z 1007.510,A 0.000,B 0.000,C 90.000,E1 271.892} C_DIS
LIN {X -0.059,Y -472.478,Z 1007.508,A 0.000,B 0.000,C 90.000,E1 271.375} C_DIS
LIN {X 0.233,Y -469.852,Z 1007.506,A 0.000,B 0.000,C 90.000,E1 271.088} C_DIS
LIN {X 0.050,Y -463.909,Z 1007.504,A 0.000,B 0.000,C 90.000,E1 270.630} C_DIS
LIN {X -0.085,Y -457.700,Z 1007.501,A 0.000,B 0.000,C 90.000,E1 270.229} C_DIS
LIN {X 0.205,Y -450.843,Z 1007.499,A 0.000,B 0.000,C 90.000,E1 269.828} C_DIS
LIN {X 0.102,Y -443.585,Z 1007.497,A 0.000,B 0.000,C 90.000,E1 269.542} C_DIS
LIN {X 0.045,Y -436.198,Z 1007.496,A 0.000,B 0.000,C 90.000,E1 269.312} C_DIS
LIN {X -0.061,Y -428.288,Z 1007.495,A 0.000,B 0.000,C 90.000,E1 269.141} C_DIS
LIN {X 0.202,Y -419.388,Z 1007.494,A 0.000,B 0.000,C 90.000,E1 268.969} C_DIS
LIN {X -0.079,Y -410.170,Z 1007.494,A 0.000,B 0.000,C 90.000,E1 268.912} C_DIS
LIN {X -0.067,Y -400.962,Z 1007.494,A 0.000,B 0.000,C 90.000,E1 268.854} C_DIS
LIN {X -0.060,Y -181.282,Z 1007.494,A 0.000,B 0.000,C 90.000,E1 268.854} C_DIS
LIN {X 0.002,Y -180.885,Z 1007.473,A 0.000,B 0.000,C 90.000,E1 265.122} C_DIS
LIN {X 0.062,Y -179.007,Z 1007.445,A 0.000,B 0.000,C 90.000,E1 260.038} C_DIS
LIN {X -0.020,Y -178.615,Z 1007.440,A 0.000,B 0.000,C 90.000,E1 259.218} C_DIS
LIN {X 0.048,Y -175.667,Z 1007.412,A 0.000,B 0.000,C 90.000,E1 254.102} C_DIS
LIN {X 0.053,Y -172.385,Z 1007.388,A 0.000,B 0.000,C 90.000,E1 249.826} C_DIS
LIN {X 0.067,Y -171.184,Z 1007.378,A 0.000,B 0.000,C 90.000,E1 248.103} C_DIS
LIN {X -0.040,Y -167.476,Z 1007.354,A 0.000,B 0.000,C 90.000,E1 243.819} C_DIS
LIN {X -0.033,Y -166.873,Z 1007.350,A 0.000,B 0.000,C 90.000,E1 242.948} C_DIS
LIN {X -0.041,Y -162.178,Z 1007.321,A 0.000,B 0.000,C 90.000,E1 237.709} C_DIS
LIN {X 0.017,Y -160.744,Z 1007.311,A 0.000,B 0.000,C 90.000,E1 235.928} C_DIS
LIN {X -0.004,Y -157.544,Z 1007.291,A 0.000,B 0.000,C 90.000,E1 232.396} C_DIS
LIN {X -0.066,Y -155.571,Z 1007.276,A 0.000,B 0.000,C 90.000,E1 229.747} C_DIS
LIN {X -0.014,Y -151.858,Z 1007.251,A 0.000,B 0.000,C 90.000,E1 225.243} C_DIS
LIN {X 0.000,Y -150.080,Z 1007.236,A 0.000,B 0.000,C 90.000,E1 222.528} C_DIS
LIN {X 0.034,Y -146.884,Z 1007.211,A 0.000,B 0.000,C 90.000,E1 217.971} C_DIS
LIN {X 0.023,Y -145.471,Z 1007.196,A 0.000,B 0.000,C 90.000,E1 215.231} C_DIS
LIN {X -0.059,Y -142.883,Z 1007.170,A 0.000,B 0.000,C 90.000,E1 210.669} C_DIS
LIN {X -0.002,Y -141.501,Z 1007.150,A 0.000,B 0.000,C 90.000,E1 206.950} C_DIS
LIN {X 0.046,Y -139.388,Z 1007.114,A 0.000,B 0.000,C 90.000,E1 200.429} C_DIS
LIN {X 0.034,Y -138.846,Z 1007.098,A 0.000,B 0.000,C 90.000,E1 197.638} C_DIS
LIN {X -0.042,Y -138.354,Z 1007.057,A 0.000,B 0.000,C 90.000,E1 190.197} C_DIS
LIN {X -0.050,Y -139.517,Z 1007.005,A 0.000,B 0.000,C 90.000,E1 180.859} C_DIS
LIN {X 0.031,Y -141.172,Z 1006.974,A 0.000,B 0.000,C 90.000,E1 175.241} C_DIS
LIN {X 0.002,Y -142.551,Z 1006.958,A 0.000,B 0.000,C 90.000,E1 172.470} C_DIS
LIN {X -0.072,Y -144.828,Z 1006.932,A 0.000,B 0.000,C 90.000,E1 167.881} C_DIS
LIN {X 0.057,Y -147.451,Z 1006.912,A 0.000,B 0.000,C 90.000,E1 164.157} C_DIS
LIN {X -0.058,Y -150.032,Z 1006.892,A 0.000,B 0.000,C 90.000,E1 160.550} C_DIS
LIN {X -0.052,Y -153.370,Z 1006.872,A 0.000,B 0.000,C 90.000,E1 156.922} C_DIS
LIN {X -0.003,Y -155.903,Z 1006.857,A 0.000,B 0.000,C 90.000,E1 154.204} C_DIS
LIN {X -0.028,Y -159.764,Z 1006.837,A 0.000,B 0.000,C 90.000,E1 150.639} C_DIS
LIN {X -0.040,Y -162.004,Z 1006.827,A 0.000,B 0.000,C 90.000,E1 148.869} C_DIS
LIN {X 0.074,Y -166.197,Z 1006.807,A 0.000,B 0.000,C 90.000,E1 145.308} C_DIS
LIN {X 0.076,Y -171.212,Z 1006.788,A 0.000,B 0.000,C 90.000,E1 141.823} C_DIS
LIN {X 0.001,Y -176.098,Z 1006.769,A 0.000,B 0.000,C 90.000,E1 138.405} C_DIS
LIN {X 0.118,Y -180.359,Z 1006.755,A 0.000,B 0.000,C 90.000,E1 135.810} C_DIS
LIN {X 0.095,Y -185.768,Z 1006.736,A 0.000,B 0.000,C 90.000,E1 132.447} C_DIS
LIN {X 0.028,Y -190.382,Z 1006.722,A 0.000,B 0.000,C 90.000,E1 129.967} C_DIS
LIN {X -0.093,Y -196.372,Z 1006.703,A 0.000,B 0.000,C 90.000,E1 126.583} C_DIS
LIN {X 0.048,Y -301.228,Z 1006.703,A 0.000,B 0.000,C 90.000,E1 126.537} C_DIS
LIN {X -0.007,Y -306.140,Z 1006.702,A 0.000,B 0.000,C 90.000,E1 126.377} C_DIS
LIN {X -0.064,Y -308.517,Z 1006.701,A 0.000,B 0.000,C 90.000,E1 126.217} C_DIS
LIN {X -0.113,Y -311.723,Z 1006.699,A 0.000,B 0.000,C 90.000,E1 125.884} C_DIS
LIN {X -0.161,Y -313.713,Z 1006.698,A 0.000,B 0.000,C 90.000,E1 125.598} C_DIS
LIN {X 0.047,Y -315.277,Z 1006.696,A 0.000,B 0.000,C 90.000,E1 125.264} C_DIS
LIN {X 0.028,Y -316.632,Z 1006.694,A 0.000,B 0.000,C 90.000,E1 124.945} C_DIS
LIN {X -0.149,Y -328.675,Z 1006.675,A 0.000,B 0.000,C 90.000,E1 121.465} C_DIS
LIN {X 0.045,Y -339.923,Z 1006.659,A 0.000,B 0.000,C 90.000,E1 118.615} C_DIS
LIN {X 0.079,Y -352.586,Z 1006.644,A 0.000,B 0.000,C 90.000,E1 115.848} C_DIS
LIN {X 0.031,Y -366.769,Z 1006.629,A 0.000,B 0.000,C 90.000,E1 113.153} C_DIS
LIN {X 0.121,Y -380.757,Z 1006.616,A 0.000,B 0.000,C 90.000,E1 110.791} C_DIS
LIN {X -0.216,Y -396.148,Z 1006.603,A 0.000,B 0.000,C 90.000,E1 108.544} C_DIS
LIN {X 0.079,Y -413.051,Z 1006.590,A 0.000,B 0.000,C 90.000,E1 106.260} C_DIS
LIN {X 0.177,Y -431.587,Z 1006.578,A 0.000,B 0.000,C 90.000,E1 104.064} C_DIS
LIN {X -0.004,Y -451.464,Z 1006.567,A 0.000,B 0.000,C 90.000,E1 102.007} C_DIS
LIN {X 0.090,Y -466.766,Z 1006.559,A 0.000,B 0.000,C 90.000,E1 100.546} C_DIS
LIN {X 0.105,Y -468.956,Z 1006.557,A 0.000,B 0.000,C 90.000,E1 100.310} C_DIS
LIN {X -0.047,Y -470.734,Z 1006.556,A 0.000,B 0.000,C 90.000,E1 100.074} C_DIS
LIN {X 0.182,Y -472.069,Z 1006.555,A 0.000,B 0.000,C 90.000,E1 99.792} C_DIS
LIN {X -0.104,Y -473.740,Z 1006.552,A 0.000,B 0.000,C 90.000,E1 99.321} C_DIS
LIN {X 0.006,Y -474.345,Z 1006.549,A 0.000,B 0.000,C 90.000,E1 98.803} C_DIS
LIN {X 0.198,Y -473.986,Z 1006.546,A 0.000,B 0.000,C 90.000,E1 98.276} C_DIS
LIN {X -0.147,Y -472.611,Z 1006.543,A 0.000,B 0.000,C 90.000,E1 97.814} C_DIS
LIN {X 0.118,Y -471.475,Z 1006.542,A 0.000,B 0.000,C 90.000,E1 97.530} C_DIS
LIN {X -0.228,Y -468.220,Z 1006.539,A 0.000,B 0.000,C 90.000,E1 97.068} C_DIS
LIN {X -0.160,Y -456.000,Z 1006.529,A 0.000,B 0.000,C 90.000,E1 95.277} C_DIS
LIN {X 0.052,Y -435.164,Z 1006.512,A 0.000,B 0.000,C 90.000,E1 92.121} C_DIS
LIN {X -0.073,Y -422.419,Z 1006.500,A 0.000,B 0.000,C 90.000,E1 90.000} C_DIS
LIN {X 0.014,Y -409.115,Z 1006.486,A 0.000,B 0.000,C 90.000,E1 87.535} C_DIS
LIN {X 0.039,Y -400.203,Z 1006.477,A 0.000,B 0.000,C 90.000,E1 85.869} C_DIS
LIN {X -0.094,Y -391.078,Z 1006.468,A 0.000,B 0.000,C 90.000,E1 84.204} C_DIS
LIN {X 0.075,Y -381.793,Z 1006.458,A 0.000,B 0.000,C 90.000,E1 82.470} C_DIS
LIN {X 0.074,Y -372.168,Z 1006.449,A 0.000,B 0.000,C 90.000,E1 80.735} C_DIS
LIN {X -0.047,Y -362.243,Z 1006.439,A 0.000,B 0.000,C 90.000,E1 78.993} C_DIS
LIN {X -0.038,Y -347.323,Z 1006.424,A 0.000,B 0.000,C 90.000,E1 76.297} C_DIS
LIN {X 0.142,Y -332.860,Z 1006.409,A 0.000,B 0.000,C 90.000,E1 73.504} C_DIS
LIN {X 0.023,Y -322.022,Z 1006.396,A 0.000,B 0.000,C 90.000,E1 71.329} C_DIS
LIN {X 0.006,Y -309.864,Z 1006.382,A 0.000,B 0.000,C 90.000,E1 68.773} C_DIS
LIN {X -0.088,Y -296.508,Z 1006.366,A 0.000,B 0.000,C 90.000,E1 65.845} C_DIS
LIN {X 0.115,Y -284.999,Z 1006.351,A 0.000,B 0.000,C 90.000,E1 63.127} C_DIS
LIN {X -0.164,Y -275.037,Z 1006.338,A 0.000,B 0.000,C 90.000,E1 60.795} C_DIS
LIN {X -0.015,Y -265.183,Z 1006.324,A 0.000,B 0.000,C 90.000,E1 58.329} C_DIS
LIN {X 0.111,Y -252.946,Z 1006.306,A 0.000,B 0.000,C 90.000,E1 55.102} C_DIS
LIN {X 0.117,Y -241.333,Z 1006.288,A 0.000,B 0.000,C 90.000,E1 51.823} C_DIS
LIN {X 0.060,Y -230.396,Z 1006.269,A 0.000,B 0.000,C 90.000,E1 48.485} C_DIS
LIN {X -0.108,Y -221.167,Z 1006.253,A 0.000,B 0.000,C 90.000,E1 45.486} C_DIS
LIN {X -0.025,Y -212.400,Z 1006.235,A 0.000,B 0.000,C 90.000,E1 42.366} C_DIS
LIN {X 0.042,Y -204.207,Z 1006.218,A 0.000,B 0.000,C 90.000,E1 39.197} C_DIS
LIN {X -0.032,Y -196.537,Z 1006.200,A 0.000,B 0.000,C 90.000,E1 36.011} C_DIS
LIN {X -0.041,Y -189.719,Z 1006.182,A 0.000,B 0.000,C 90.000,E1 32.752} C_DIS
LIN {X 0.060,Y -183.683,Z 1006.164,A 0.000,B 0.000,C 90.000,E1 29.411} C_DIS
LIN {X -0.092,Y -178.462,Z 1006.145,A 0.000,B 0.000,C 90.000,E1 26.104} C_DIS
LIN {X -0.049,Y -174.006,Z 1006.126,A 0.000,B 0.000,C 90.000,E1 22.695} C_DIS
LIN {X -0.059,Y -170.220,Z 1006.107,A 0.000,B 0.000,C 90.000,E1 19.268} C_DIS
LIN {X 0.062,Y -166.512,Z 1006.083,A 0.000,B 0.000,C 90.000,E1 14.898} C_DIS
LIN {X 0.025,Y -163.835,Z 1006.059,A 0.000,B 0.000,C 90.000,E1 10.546} C_DIS
LIN {X 0.068,Y -161.764,Z 1006.020,A 0.000,B 0.000,C 90.000,E1 3.498} C_DIS
LIN {X 0.073,Y -163.126,Z 1005.963,A 0.000,B 0.000,C 90.000,E1 353.337} C_DIS
LIN {X -0.025,Y -165.833,Z 1005.934,A 0.000,B 0.000,C 90.000,E1 348.105} C_DIS
LIN {X -0.006,Y -169.271,Z 1005.910,A 0.000,B 0.000,C 90.000,E1 343.740} C_DIS
LIN {X -0.059,Y -172.845,Z 1005.890,A 0.000,B 0.000,C 90.000,E1 340.296} C_DIS
LIN {X -0.004,Y -177.270,Z 1005.871,A 0.000,B 0.000,C 90.000,E1 336.847} C_DIS
LIN {X -0.032,Y -182.503,Z 1005.852,A 0.000,B 0.000,C 90.000,E1 333.461} C_DIS
LIN {X 0.063,Y -188.533,Z 1005.834,A 0.000,B 0.000,C 90.000,E1 330.078} C_DIS
LIN {X 0.008,Y -195.257,Z 1005.815,A 0.000,B 0.000,C 90.000,E1 326.786} C_DIS
LIN {X -0.040,Y -202.523,Z 1005.797,A 0.000,B 0.000,C 90.000,E1 323.543} C_DIS
LIN {X -0.104,Y -210.419,Z 1005.780,A 0.000,B 0.000,C 90.000,E1 320.356} C_DIS
LIN {X 0.050,Y -219.786,Z 1005.760,A 0.000,B 0.000,C 90.000,E1 316.782} C_DIS
LIN {X -0.019,Y -230.039,Z 1005.741,A 0.000,B 0.000,C 90.000,E1 313.338} C_DIS
LIN {X -0.080,Y -235.174,Z 1005.732,A 0.000,B 0.000,C 90.000,E1 311.838} C_DIS
LIN {X 0.076,Y -242.522,Z 1005.722,A 0.000,B 0.000,C 90.000,E1 309.930} C_DIS
LIN {X 0.039,Y -250.733,Z 1005.712,A 0.000,B 0.000,C 90.000,E1 308.096} C_DIS
LIN {X 0.015,Y -261.730,Z 1005.700,A 0.000,B 0.000,C 90.000,E1 305.931} C_DIS
LIN {X 0.125,Y -277.988,Z 1005.684,A 0.000,B 0.000,C 90.000,E1 303.086} C_DIS
LIN {X -0.014,Y -293.314,Z 1005.671,A 0.000,B 0.000,C 90.000,E1 300.718} C_DIS
LIN {X 0.032,Y -311.971,Z 1005.656,A 0.000,B 0.000,C 90.000,E1 298.052} C_DIS
LIN {X 0.085,Y -324.698,Z 1005.647,A 0.000,B 0.000,C 90.000,E1 296.437} C_DIS
LIN {X -0.003,Y -338.381,Z 1005.638,A 0.000,B 0.000,C 90.000,E1 294.899} C_DIS
LIN {X -0.024,Y -360.478,Z 1005.626,A 0.000,B 0.000,C 90.000,E1 292.642} C_DIS
LIN {X -0.126,Y -379.769,Z 1005.616,A 0.000,B 0.000,C 90.000,E1 290.844} C_DIS
LIN {X -0.008,Y -393.434,Z 1005.609,A 0.000,B 0.000,C 90.000,E1 289.577} C_DIS
LIN {X 0.144,Y -406.843,Z 1005.602,A 0.000,B 0.000,C 90.000,E1 288.308} C_DIS
LIN {X -0.069,Y -414.593,Z 1005.598,A 0.000,B 0.000,C 90.000,E1 287.583} C_DIS
LIN {X -0.034,Y -422.139,Z 1005.593,A 0.000,B 0.000,C 90.000,E1 286.804} C_DIS
LIN {X 0.060,Y -431.934,Z 1005.587,A 0.000,B 0.000,C 90.000,E1 285.733} C_DIS
LIN {X 0.076,Y -441.218,Z 1005.581,A 0.000,B 0.000,C 90.000,E1 284.662} C_DIS
LIN {X 0.201,Y -449.960,Z 1005.576,A 0.000,B 0.000,C 90.000,E1 283.592} C_DIS
LIN {X -0.123,Y -458.063,Z 1005.570,A 0.000,B 0.000,C 90.000,E1 282.591} C_DIS
LIN {X -0.194,Y -463.626,Z 1005.566,A 0.000,B 0.000,C 90.000,E1 281.827} C_DIS
LIN {X -0.007,Y -470.296,Z 1005.560,A 0.000,B 0.000,C 90.000,E1 280.782} C_DIS
LIN {X 0.022,Y -474.721,Z 1005.556,A 0.000,B 0.000,C 90.000,E1 280.018} C_DIS
LIN {X 0.007,Y -478.530,Z 1005.551,A 0.000,B 0.000,C 90.000,E1 279.265} C_DIS
LIN {X 0.025,Y -481.665,Z 1005.547,A 0.000,B 0.000,C 90.000,E1 278.511} C_DIS
LIN {X 0.184,Y -483.482,Z 1005.544,A 0.000,B 0.000,C 90.000,E1 277.992} C_DIS
LIN {X -0.121,Y -484.994,Z 1005.542,A 0.000,B 0.000,C 90.000,E1 277.530} C_DIS
LIN {X 0.124,Y -486.303,Z 1005.539,A 0.000,B 0.000,C 90.000,E1 277.004} C_DIS
LIN {X -0.169,Y -487.343,Z 1005.536,A 0.000,B 0.000,C 90.000,E1 276.543} C_DIS
LIN {X -0.021,Y -488.172,Z 1005.534,A 0.000,B 0.000,C 90.000,E1 276.030} C_DIS
LIN {X 0.188,Y -488.707,Z 1005.531,A 0.000,B 0.000,C 90.000,E1 275.511} C_DIS
LIN {X -0.086,Y -488.893,Z 1005.528,A 0.000,B 0.000,C 90.000,E1 275.049} C_DIS
LIN {X 0.128,Y -488.616,Z 1005.525,A 0.000,B 0.000,C 90.000,E1 274.531} C_DIS
LIN {X -0.147,Y -487.917,Z 1005.523,A 0.000,B 0.000,C 90.000,E1 274.069} C_DIS
LIN {X 0.029,Y -486.642,Z 1005.520,A 0.000,B 0.000,C 90.000,E1 273.555} C_DIS
LIN {X 0.231,Y -484.798,Z 1005.517,A 0.000,B 0.000,C 90.000,E1 273.037} C_DIS
LIN {X -0.084,Y -482.216,Z 1005.514,A 0.000,B 0.000,C 90.000,E1 272.579} C_DIS
LIN {X 0.070,Y -478.946,Z 1005.512,A 0.000,B 0.000,C 90.000,E1 272.064} C_DIS
LIN {X 0.221,Y -474.742,Z 1005.509,A 0.000,B 0.000,C 90.000,E1 271.547} C_DIS
LIN {X -0.138,Y -469.597,Z 1005.506,A 0.000,B 0.000,C 90.000,E1 271.088} C_DIS
LIN {X -0.189,Y -466.833,Z 1005.505,A 0.000,B 0.000,C 90.000,E1 270.859} C_DIS
LIN {X -0.049,Y -460.789,Z 1005.502,A 0.000,B 0.000,C 90.000,E1 270.401} C_DIS
LIN {X 0.095,Y -454.310,Z 1005.500,A 0.000,B 0.000,C 90.000,E1 270.000} C_DIS
LIN {X -0.199,Y -447.418,Z 1005.498,A 0.000,B 0.000,C 90.000,E1 269.714} C_DIS
LIN {X -0.033,Y -440.190,Z 1005.497,A 0.000,B 0.000,C 90.000,E1 269.427} C_DIS
LIN {X 0.094,Y -432.540,Z 1005.496,A 0.000,B 0.000,C 90.000,E1 269.198} C_DIS
LIN {X 0.182,Y -424.187,Z 1005.495,A 0.000,B 0.000,C 90.000,E1 269.026} C_DIS
LIN {X 0.174,Y -415.543,Z 1005.494,A 0.000,B 0.000,C 90.000,E1 268.912} C_DIS
LIN {X -0.161,Y -401.672,Z 1005.494,A 0.000,B 0.000,C 90.000,E1 268.854} C_DIS
LIN {X 0.175,Y -399.487,Z 1005.493,A 0.000,B 0.000,C 90.000,E1 268.797} C_DIS
LIN {X 0.051,Y -181.278,Z 1005.493,A 0.000,B 0.000,C 90.000,E1 268.797} C_DIS
LIN {X -0.066,Y -180.882,Z 1005.473,A 0.000,B 0.000,C 90.000,E1 265.122} C_DIS
LIN {X -0.007,Y -179.002,Z 1005.445,A 0.000,B 0.000,C 90.000,E1 260.038} C_DIS
LIN {X 0.087,Y -178.599,Z 1005.440,A 0.000,B 0.000,C 90.000,E1 259.162} C_DIS
LIN {X -0.020,Y -175.652,Z 1005.412,A 0.000,B 0.000,C 90.000,E1 254.102} C_DIS
LIN {X -0.014,Y -172.370,Z 1005.388,A 0.000,B 0.000,C 90.000,E1 249.826} C_DIS
LIN {X 0.001,Y -171.162,Z 1005.378,A 0.000,B 0.000,C 90.000,E1 248.103} C_DIS
LIN {X 0.044,Y -167.461,Z 1005.354,A 0.000,B 0.000,C 90.000,E1 243.768} C_DIS
LIN {X -0.022,Y -166.857,Z 1005.350,A 0.000,B 0.000,C 90.000,E1 242.922} C_DIS
LIN {X 0.042,Y -162.842,Z 1005.325,A 0.000,B 0.000,C 90.000,E1 238.535} C_DIS
LIN {X 0.018,Y -161.526,Z 1005.315,A 0.000,B 0.000,C 90.000,E1 236.786} C_DIS
LIN {X 0.057,Y -157.526,Z 1005.291,A 0.000,B 0.000,C 90.000,E1 232.351} C_DIS
LIN {X -0.010,Y -155.551,Z 1005.276,A 0.000,B 0.000,C 90.000,E1 229.703} C_DIS
LIN {X -0.076,Y -151.842,Z 1005.251,A 0.000,B 0.000,C 90.000,E1 225.243} C_DIS
LIN {X -0.061,Y -150.061,Z 1005.236,A 0.000,B 0.000,C 90.000,E1 222.528} C_DIS
LIN {X -0.027,Y -146.871,Z 1005.211,A 0.000,B 0.000,C 90.000,E1 217.971} C_DIS
LIN {X -0.037,Y -145.456,Z 1005.196,A 0.000,B 0.000,C 90.000,E1 215.231} C_DIS
LIN {X 0.076,Y -142.873,Z 1005.170,A 0.000,B 0.000,C 90.000,E1 210.590} C_DIS
LIN {X 0.001,Y -141.490,Z 1005.150,A 0.000,B 0.000,C 90.000,E1 206.924} C_DIS
LIN {X -0.013,Y -139.385,Z 1005.113,A 0.000,B 0.000,C 90.000,E1 200.429} C_DIS
LIN {X -0.024,Y -138.840,Z 1005.098,A 0.000,B 0.000,C 90.000,E1 197.638} C_DIS
LIN {X 0.036,Y -138.354,Z 1005.056,A 0.000,B 0.000,C 90.000,E1 190.141} C_DIS
LIN {X 0.031,Y -139.521,Z 1005.005,A 0.000,B 0.000,C 90.000,E1 180.802} C_DIS
LIN {X -0.028,Y -141.183,Z 1004.974,A 0.000,B 0.000,C 90.000,E1 175.241} C_DIS
LIN {X -0.057,Y -142.561,Z 1004.958,A 0.000,B 0.000,C 90.000,E1 172.470} C_DIS
LIN {X 0.009,Y -144.843,Z 1004.932,A 0.000,B 0.000,C 90.000,E1 167.825} C_DIS
LIN {X -0.005,Y -147.467,Z 1004.912,A 0.000,B 0.000,C 90.000,E1 164.157} C_DIS
LIN {X 0.022,Y -150.051,Z 1004.892,A 0.000,B 0.000,C 90.000,E1 160.496} C_DIS
LIN {X 0.027,Y -153.395,Z 1004.872,A 0.000,B 0.000,C 90.000,E1 156.869} C_DIS
LIN {X 0.073,Y -155.925,Z 1004.857,A 0.000,B 0.000,C 90.000,E1 154.152} C_DIS
LIN {X 0.048,Y -159.791,Z 1004.837,A 0.000,B 0.000,C 90.000,E1 150.589} C_DIS
LIN {X 0.033,Y -162.033,Z 1004.827,A 0.000,B 0.000,C 90.000,E1 148.820} C_DIS
LIN {X 0.008,Y -166.227,Z 1004.807,A 0.000,B 0.000,C 90.000,E1 145.308} C_DIS
LIN {X 0.009,Y -171.244,Z 1004.788,A 0.000,B 0.000,C 90.000,E1 141.823} C_DIS
LIN {X -0.068,Y -176.132,Z 1004.769,A 0.000,B 0.000,C 90.000,E1 138.405} C_DIS
LIN {X 0.048,Y -180.399,Z 1004.755,A 0.000,B 0.000,C 90.000,E1 135.810} C_DIS
LIN {X 0.024,Y -185.806,Z 1004.736,A 0.000,B 0.000,C 90.000,E1 132.447} C_DIS
LIN {X 0.079,Y -190.424,Z 1004.722,A 0.000,B 0.000,C 90.000,E1 129.930} C_DIS
LIN {X 0.028,Y -196.305,Z 1004.703,A 0.000,B 0.000,C 90.000,E1 126.583} C_DIS
LIN {X 0.009,Y -300.927,Z 1004.703,A 0.000,B 0.000,C 90.000,E1 126.583} C_DIS
LIN {X 0.117,Y -303.594,Z 1004.703,A 0.000,B 0.000,C 90.000,E1 126.503} C_DIS
LIN {X 0.071,Y -309.028,Z 1004.701,A 0.000,B 0.000,C 90.000,E1 126.171} C_DIS
LIN {X -0.046,Y -312.019,Z 1004.699,A 0.000,B 0.000,C 90.000,E1 125.851} C_DIS
LIN {X 0.076,Y -313.999,Z 1004.697,A 0.000,B 0.000,C 90.000,E1 125.518} C_DIS
LIN {X -0.058,Y -315.545,Z 1004.696,A 0.000,B 0.000,C 90.000,E1 125.231} C_DIS
LIN {X 0.060,Y -317.855,Z 1004.692,A 0.000,B 0.000,C 90.000,E1 124.565} C_DIS
LIN {X 0.010,Y -328.843,Z 1004.674,A 0.000,B 0.000,C 90.000,E1 121.386} C_DIS
LIN {X 0.046,Y -340.116,Z 1004.659,A 0.000,B 0.000,C 90.000,E1 118.565} C_DIS
LIN {X 0.094,Y -352.805,Z 1004.643,A 0.000,B 0.000,C 90.000,E1 115.796} C_DIS
LIN {X 0.204,Y -367.015,Z 1004.628,A 0.000,B 0.000,C 90.000,E1 113.078} C_DIS
LIN {X 0.164,Y -381.031,Z 1004.615,A 0.000,B 0.000,C 90.000,E1 110.737} C_DIS
LIN {X -0.034,Y -396.451,Z 1004.603,A 0.000,B 0.000,C 90.000,E1 108.471} C_DIS
LIN {X 0.150,Y -413.386,Z 1004.590,A 0.000,B 0.000,C 90.000,E1 106.205} C_DIS
LIN {X -0.155,Y -431.956,Z 1004.578,A 0.000,B 0.000,C 90.000,E1 104.064} C_DIS
LIN {X 0.116,Y -451.848,Z 1004.566,A 0.000,B 0.000,C 90.000,E1 101.951} C_DIS
LIN {X -0.223,Y -467.145,Z 1004.558,A 0.000,B 0.000,C 90.000,E1 100.546} C_DIS
LIN {X -0.205,Y -469.232,Z 1004.557,A 0.000,B 0.000,C 90.000,E1 100.310} C_DIS
LIN {X 0.105,Y -470.939,Z 1004.556,A 0.000,B 0.000,C 90.000,E1 100.018} C_DIS
LIN {X -0.129,Y -472.222,Z 1004.554,A 0.000,B 0.000,C 90.000,E1 99.792} C_DIS
LIN {X 0.053,Y -473.811,Z 1004.552,A 0.000,B 0.000,C 90.000,E1 99.265} C_DIS
LIN {X 0.164,Y -474.347,Z 1004.549,A 0.000,B 0.000,C 90.000,E1 98.746} C_DIS
LIN {X -0.112,Y -473.920,Z 1004.546,A 0.000,B 0.000,C 90.000,E1 98.276} C_DIS
LIN {X 0.013,Y -472.468,Z 1004.543,A 0.000,B 0.000,C 90.000,E1 97.757} C_DIS
LIN {X -0.189,Y -471.284,Z 1004.542,A 0.000,B 0.000,C 90.000,E1 97.530} C_DIS
LIN {X -0.013,Y -467.983,Z 1004.539,A 0.000,B 0.000,C 90.000,E1 97.004} C_DIS
LIN {X -0.009,Y -455.770,Z 1004.529,A 0.000,B 0.000,C 90.000,E1 95.220} C_DIS
LIN {X 0.191,Y -434.960,Z 1004.512,A 0.000,B 0.000,C 90.000,E1 92.064} C_DIS
LIN {X 0.056,Y -422.239,Z 1004.500,A 0.000,B 0.000,C 90.000,E1 89.943} C_DIS
LIN {X 0.135,Y -408.939,Z 1004.486,A 0.000,B 0.000,C 90.000,E1 87.478} C_DIS
LIN {X 0.154,Y -400.016,Z 1004.477,A 0.000,B 0.000,C 90.000,E1 85.812} C_DIS
LIN {X 0.067,Y -389.349,Z 1004.466,A 0.000,B 0.000,C 90.000,E1 83.856} C_DIS
